// Else if own TU data index is free
ELSIF ZoneData.TransportControlData.TU_DataIndex = 0 THEN
	// Move TU data index from previous to own zone
	mTU_DataIndex := F_MoveTU_DataIndex(
							eFunctionNumber := PrevTransportData.eFunctionNumber,
							mZoneNumber     := PrevTransportData.ZoneNumber);

	// Update zone data
	ZoneData.TransportControlData.TU_DataIndex := mTU_DataIndex;
	ZoneData.TransportControlData.DataPresent := mTU_DataIndex <> 0;
	ZoneData.TransportControlData.NumberOfPresentTUs := 1;

	// Check if the TU data index is valid - if not, create a debug message
	IF mTU_DataIndex < 0 OR mTU_DataIndex > Conveyor.NUMBER_OF_TU_DATA THEN
		// debug message: '11-001-0095-01-1,  TU_DataIndex is out of range,  TU_DataIndex = 5000,  range = 0..1979'
		DebugMsg:= '';
		DebugMsg:= CONCAT(DebugMsg, Param.rSettings.ZoneName);
		DebugMsg:= CONCAT(DebugMsg, ',  TU_DataIndex is out of range');
		DebugMsg:= CONCAT(DebugMsg, DebugTextBlocks.TU_DATA_INDEX);
		DebugMsg:= CONCAT(DebugMsg, DINT_TO_STRING(mTU_DataIndex));
		DebugMsg:= CONCAT(DebugMsg, DebugTextBlocks.RANGE);
		DebugMsg:= CONCAT(DebugMsg, DINT_TO_STRING(Conveyor.NUMBER_OF_TU_DATA));
		fbDebugMsg.M_SendErrorMsg(DebugMsg);				  
		
	// Else if a valid TU data index is available check whether the index matches the expected position.
	// If not the TU index is incorrectly linked to multiple positions at the same time.
	ELSIF mTU_DataIndex <> 0 THEN
		mCurrentFunctionNumber := TU_Table.TU_DataTable[mTU_DataIndex].CurrentFunctionNumber;
		mCurrentZoneNumber := TU_Table.TU_DataTable[mTU_DataIndex].CurrentZoneNumber;
		
		// If function and zone number is valid
		IF mCurrentFunctionNumber <> 0 AND mCurrentZoneNumber <> 0 THEN
			// If current TU position is not previous zone
			IF mCurrentFunctionNumber <> PrevTransportData.eFunctionNumber OR mCurrentZoneNumber <> PrevTransportData.ZoneNumber THEN
				// debug message: '11-001-0095-01-1,  incorrectly linked TU_DataIndex to current TU position,  expected = 11-222-3333-44-5,  current = 99-9999-1979-01-9'
				DebugMsg:= '';
				DebugMsg:= CONCAT(DebugMsg, Param.rSettings.ZoneName);
				DebugMsg:= CONCAT(DebugMsg, ',  incorrectly linked TU_DataIndex to current TU position');
				DebugMsg:= CONCAT(DebugMsg, DebugTextBlocks.EXPECTED);
				DebugMsg:= CONCAT(DebugMsg, F_GetFunctionName(
												eFunctionNumber := PrevTransportData.eFunctionNumber,
												ZoneNumber := PrevTransportData.ZoneNumber));
				DebugMsg:= CONCAT(DebugMsg, DebugTextBlocks.CURRENT);
				DebugMsg:= CONCAT(DebugMsg, F_GetFunctionName(
												eFunctionNumber := mCurrentFunctionNumber,
												ZoneNumber := mCurrentZoneNumber));
				DebugMsg:= CONCAT(DebugMsg, F_CreateTU_DataString(mTU_DataIndex));
				fbDebugMsg.M_SendErrorMsg(DebugMsg);				  
			END_IF
		END_IF

		// Update currrent TU position
		TU_Table.TU_DataTable[mTU_DataIndex].CurrentFunctionNumber := Param.reFunctionNumber;
		TU_Table.TU_DataTable[mTU_DataIndex].CurrentZoneNumber := Param.ZoneNumber;
	END_IF

ELSE
	// Own TU data index is already used
	mTU_DataIndex := ZoneData.TransportControlData.TU_DataIndex;

	// Set error TU data index is not free
	F_SetError(
		ErrorType := E_ErrorType.ERROR,
		ErrorParam:= CONCAT('TU-DataIndex = ', DINT_TO_STRING(mTU_DataIndex)),
		ErrorMsg  := E_ErrorConv.TU_DATA_INDEX_NOT_FREE,
		ErrorData := ErrorData);
	
	// debug message: '11-001-0095-01-1,  own TU data index not free,  TU_DataIndex = 12345,  TuID = 112233,  AssignmentID = 12345678'
	DebugMsg:= '';
	DebugMsg:= CONCAT(DebugMsg, Param.rSettings.ZoneName);
	DebugMsg:= CONCAT(DebugMsg, ',  own TU data index not free');
	DebugMsg:= CONCAT(DebugMsg, F_CreateTU_DataString(mTU_DataIndex));
	fbDebugMsg.M_SendErrorMsg(DebugMsg);				  
	
	// Update number of present TUs
	ZoneData.TransportControlData.NumberOfPresentTUs := 1;
END_IF
{warning restore C0371}
END_METHOD

// Requests the routing service to retrieve next partner
METHOD PROTECTED M_RequestNext
(**************************************************************************************
 *  Application     :   BoxControl Framework
 *  Revision date   :   $Date: 2021-04-10 12:07:10 +0200 (lör, 10 apr 2021) $
 *  Author          :   CDC
 * ------------------------------------------------------------------------------------
 *  © Swisslog AG
 *  Swisslog is not liable for any usage of this source code that is not agreed 
 *  on between Swisslog and the other party. The mandatory legal liability remains 
 *  unaffected.
 * ------------------------------------------------------------------------------------
 *  Revision History: 
 *
 *  VERSION DATE         INITIALS     DESCRIPTION
 *  0.0     DD.MM.YYYY   (name)       (explain customized modifications)
 *
 **************************************************************************************)
VAR_INPUT
END_VAR
{warning disable C0371}
// If no next zone or function is available
IF NextTransportData.eFunctionNumber = E_FunctionNumber.F_BEGIN_FUNCTION AND
   Param.reNextFunctionNumber = E_FunctionNumber.F_BEGIN_FUNCTION THEN	
	fbRoutingServiceRetry(IN := FALSE);
	TransportTrspDataReq.RequestNextTransportData := TRUE;

// If the routing update is enable	
ELSIF Param.rSettings.EnableRoutingUpdate THEN
	// If the next function ist not fix
	IF Param.reSetFuncNextFuncNumber = E_FunctionNumber.F_BEGIN_FUNCTION
	   AND NOT NextTransportData.rTransportControlData.TransportActive THEN
		// If the transport does not start in a reasonable time, initiate routing update
		IF ZoneData.TransportControlData.eHandOverState = E_HandOverState.IDLE OR
		   ZoneData.TransportControlData.eHandOverState = E_HandOverState.READY THEN
			fbRoutingServiceRetry(IN := TRUE, PT := RECALL_SERVICE_TIMEOUT);
			IF fbRoutingServiceRetry.Q THEN
				fbRoutingServiceRetry(IN := FALSE);
				TransportTrspDataReq.DeleteNextTransportData := TRUE;
				TransportTrspDataReq.RequestNextTransportData := TRUE;
			END_IF
		ELSE
			fbRoutingServiceRetry(IN := FALSE);
		END_IF
	ELSE
		fbRoutingServiceRetry(IN := FALSE);
	END_IF
END_IF
{warning restore C0371}
END_METHOD

// Requests the merging service to retrieve prev partner
METHOD PROTECTED M_RequestPrev
(**************************************************************************************
 *  Application     :   BoxControl Framework
 *  Revision date   :   $Date: 2021-04-10 12:07:10 +0200 (lör, 10 apr 2021) $
 *  Author          :   CDC
 * ------------------------------------------------------------------------------------
 *  © Swisslog AG
 *  Swisslog is not liable for any usage of this source code that is not agreed 
 *  on between Swisslog and the other party. The mandatory legal liability remains 
 *  unaffected.
 * ------------------------------------------------------------------------------------
 *  Revision History: 
 *
 *  VERSION DATE         INITIALS     DESCRIPTION
 *  0.0     DD.MM.YYYY   (name)       (explain customized modifications)
 *
 **************************************************************************************)
VAR_INPUT
END_VAR
{warning disable C0371}
// If no previous zone or function is available
IF PrevTransportData.eFunctionNumber = E_FunctionNumber.F_BEGIN_FUNCTION AND
   Param.rePrevFunctionNumber = E_FunctionNumber.F_BEGIN_FUNCTION THEN	
	fbMergingServiceRetry(IN := FALSE);
	TransportTrspDataReq.RequestPrevTransportData := TRUE;


// If the previous function ist not fix
ELSIF Param.reSetFuncPrevFuncNumber = E_FunctionNumber.F_BEGIN_FUNCTION
   AND NOT PrevTransportData.rTransportControlData.TransportActive THEN
	// If the transport does not start in a reasonable time, initiate merging update
	IF ZoneData.TransportControlData.eTakeOverState = E_TakeOverState.IDLE OR
	   ZoneData.TransportControlData.eTakeOverState = E_TakeOverState.READY THEN
		fbMergingServiceRetry(IN := TRUE, PT := RECALL_SERVICE_TIMEOUT);
		IF fbMergingServiceRetry.Q THEN
			fbMergingServiceRetry(IN := FALSE);
			TransportTrspDataReq.DeletePrevTransportData := TRUE;
			TransportTrspDataReq.RequestPrevTransportData := TRUE;
		END_IF
	END_IF
END_IF
{warning restore C0371}
END_METHOD

METHOD M_SelectSensor : BOOL
(**************************************************************************************
 *  Application     :   BoxControl Framework
 *  Revision date   :   $Date: 2021-04-10 12:07:10 +0200 (lör, 10 apr 2021) $
 *  Author          :   CDC
 * ------------------------------------------------------------------------------------
 *  © Swisslog AG
 *  Swisslog is not liable for any usage of this source code that is not agreed 
 *  on between Swisslog and the other party. The mandatory legal liability remains 
 *  unaffected.
 * ------------------------------------------------------------------------------------
 *  Revision History: 
 *
 *  VERSION DATE         INITIALS     DESCRIPTION
 *  0.0     DD.MM.YYYY   (name)       (explain customized modifications)
 *
 **************************************************************************************)
VAR_INPUT
END_VAR
{warning disable C0371}
IF ZoneData.AddOn.Orders.UseOwnSensor OR NOT Param.rSettings.EnableAddOnSensor THEN
    ZoneOccupiedSignal := ZoneOccupied;
ELSE
    ZoneOccupiedSignal := ZoneData.AddOn.Orders.AddOnSensor;
END_IF
{warning restore C0371}
END_METHOD

// Starts the tracking of the leading edge arriving from prev zone
METHOD PROTECTED M_StartPositionTracking
(**************************************************************************************
 *  Application     :   BoxControl Framework
 *  Revision date   :   $Date: 2021-04-10 12:07:10 +0200 (lör, 10 apr 2021) $
 *  Author          :   CDC
 * ------------------------------------------------------------------------------------
 *  © Swisslog AG
 *  Swisslog is not liable for any usage of this source code that is not agreed 
 *  on between Swisslog and the other party. The mandatory legal liability remains 
 *  unaffected.
 * ------------------------------------------------------------------------------------
 *  Revision History: 
 *
 *  VERSION DATE         INITIALS     DESCRIPTION
 *  0.0     DD.MM.YYYY   (name)       (explain customized modifications)
 *
 **************************************************************************************)
VAR
	PresetDistance     			: DINT; // Present distance for tracking leading edge
END_VAR

// Set preset distance based on available previous position data	
IF PrevTransportData.rTransportControlData.TU_LeadingEdgePos <> 0 THEN
	PresetDistance := -(UINT_TO_DINT(PrevTransportParam.ZoneLength) - PrevTransportData.rTransportControlData.TU_LeadingEdgePos);
ELSE
	PresetDistance := -(UINT_TO_DINT(PrevTransportParam.ZoneEndLength) - PrevTransportParam.StopDelayDistance);
END_IF

// Start tracking 
fbTrackingLeadingEdge(Run := FALSE);

fbTrackingLeadingEdge(Run	:= TRUE,
		EncoderValueInc 	:= EncoderValue,
		MaxEncoderValueInc	:= MaxEncoderValue,
		RateIncPerMM		:= 1,
		SetPoint			:= UINT_TO_DINT(16#FFFF),
		StartPoint			:= PresetDistance);
END_METHOD

// Calculates the distance, the TU must at least travel to be considered plausible
METHOD PROTECTED M_TakeoverPlausibleDistance : DINT
(**************************************************************************************
 *  Application     :   BoxControl Framework
 *  Revision date   :   $Date: 2021-04-10 12:07:10 +0200 (lör, 10 apr 2021) $
 *  Author          :   CDC
 * ------------------------------------------------------------------------------------
 *  © Swisslog AG
 *  Swisslog is not liable for any usage of this source code that is not agreed 
 *  on between Swisslog and the other party. The mandatory legal liability remains 
 *  unaffected.
 * ------------------------------------------------------------------------------------
 *  Revision History: 
 *
 *  VERSION DATE         INITIALS     DESCRIPTION
 *  0.0     DD.MM.YYYY   (name)       (explain customized modifications)
 *
 **************************************************************************************)
VAR
	Temp		: DINT		:= 0;
END_VAR

// valid value given from config -> use this
IF Param.rSettings.TakeoverPlausibilityDistance <> 0 THEN
	M_TakeoverPlausibleDistance := Param.rSettings.TakeoverPlausibilityDistance;
	RETURN;
END_IF

// no, calculate it:
// distance between TU's leading edge to the border of the prev zone 
Temp:= PrevTransportParam.ZoneEndLength - PrevTransportParam.StopDelayDistance;

// adding the distance from begin of own zone to the sensor
Temp:= Temp + UINT_TO_DINT(TransportParam.ZoneLength) - TransportParam.ZoneEndLength;

// return reduced value to give space for tolerance
M_TakeoverPlausibleDistance:= Temp - DIST_TO_OCCUPIED;
END_METHOD

END_FUNCTION_BLOCK

// ---- 20_Product/10_BCF/11_Conv/12_E_Functions/10_Helper/F_AckAddon.TcPOU
FUNCTION F_AckAddon : BOOL
(**************************************************************************************
 * 	Application		:	BoxControl Framework
 *	Revision		:	$Revision: 404529 $
 *	Revision date	:	$Date: 2018-04-23 08:21:38 +0200 (Mo., 23 Apr 2018) $
 *	Last changed by	:	$Author: b7bolm $
 *	URL				:	$URL: http://almscdc.swisslog.com/repo/SWPD/Development/BoxControlFramework/20_Release/trunk/01_Software/BCF/BCF/JumpStart/20_Product/10_App/12_E_Functions/10_Lib/10_Conv/10_Functions/F_AckAddon.TcPOU $
 *
 *	Purpose			:	Send acknowledge to an addon.
 *						Return Ack successful.
 *
 * ------------------------------------------------------------------------------------
 *	Copyright Swisslog [IP AG], Switzerland. All rights reserved.
 * 
 * ------------------------------------------------------------------------------------
 *	
 * 	Revision History: 
 *
 * 	VERSION			DATE			INITIALS			DESCRIPTION
 *	0.1				01.01.2001		swl					Example
 *
 **************************************************************************************)
VAR_INPUT
	eFunctionNumber			: E_FunctionNumber; // Element function Number
END_VAR



// Check if function number is valid
IF eFunctionNumber > E_FunctionNumber.F_BEGIN_FUNCTION AND
   eFunctionNumber < E_FunctionNumber.F_END_FUNCTION THEN

	F_AckAddon := __ISVALIDREF(FunctionRegistry[eFunctionNumber].rFunction);
	
	// Check reference is valid
	IF F_AckAddon THEN
   		// Send Ack command
   		FunctionRegistry[eFunctionNumber].rFunction.M_AddOnAck();
	END_IF
END_IF

END_FUNCTION

// ---- 20_Product/10_BCF/11_Conv/12_E_Functions/10_Helper/F_CheckDestination.TcPOU
FUNCTION F_CheckDestination : BOOL
(**************************************************************************************
 * 	Application		:	BoxControl Framework
 *	Revision		:	$Revision: 404529 $
 *	Revision date	:	$Date: 2018-04-23 08:21:38 +0200 (Mo., 23 Apr 2018) $
 *	Last changed by	:	$Author: b7bolm $
 *	URL				:	$URL: http://almscdc.swisslog.com/repo/SWPD/Development/BoxControlFramework/20_Release/trunk/01_Software/BCF/BCF/JumpStart/20_Product/10_App/12_E_Functions/10_Lib/10_Conv/10_Functions/F_CheckDestination.TcPOU $
 *
 *	Purpose			:	Check if TU on a position consists of the desired destination
 ç						Result True = Destination found
 *
 * ------------------------------------------------------------------------------------
 *	Copyright Swisslog [IP AG], Switzerland. All rights reserved.
 * 
 * ------------------------------------------------------------------------------------
 *	
 * 	Revision History: 
 *
 * 	VERSION			DATE			INITIALS			DESCRIPTION
 *	0.1				01.01.2001		swl					Example
 *
 **************************************************************************************)
VAR_INPUT
	eFunctionNumber		: E_FunctionNumber; // Function number
	ZoneNumber			: INT; // ZoneNumber
	DestFunctionNumber	: E_FunctionNumber; // Destination function number
	DestZoneNumber		: INT; // Destination zone number
END_VAR

VAR
	TU_DataIndex		: DINT;
	Idx					: INT;
END_VAR

// Init
F_CheckDestination := FALSE;

// Validate inputs
IF eFunctionNumber > E_FunctionNumber.F_BEGIN_FUNCTION AND
   eFunctionNumber < E_FunctionNumber.F_END_FUNCTION AND
   ZoneNumber > 0 AND
   ZoneNumber <= Conveyor.NUMBER_OF_ZONES_PER_FUNCTION THEN
   	// If zone is valid and consists of a TU-Data index
	IF __ISVALIDREF(FunctionRegistry[eFunctionNumber].Zone[ZoneNumber].refZoneData) THEN
		TU_DataIndex := FunctionRegistry[eFunctionNumber].Zone[ZoneNumber].refZoneData.TransportControlData.TU_DataIndex;
		
		IF TU_DataIndex > 0 THEN
			// Search for destination
			FOR Idx := 1 TO Conveyor.NUMBER_OF_DESTINATIONS DO
				IF TU_DataTable[TU_DataIndex].Destination[Idx].eFunctionNumber = DestFunctionNumber AND
				   TU_DataTable[TU_DataIndex].Destination[Idx].ZoneNumber = DestZoneNumber THEN
				   // Destination found
				   F_CheckDestination := TRUE;
				   EXIT;
				END_IF
			END_FOR
		END_IF
	END_IF
END_IF

END_FUNCTION

// ---- 20_Product/10_BCF/11_Conv/12_E_Functions/10_Helper/F_GetAdjacentTransportData.TcPOU
FUNCTION F_GetAdjacentTransportData : ST_TransportData
(**************************************************************************************
 * 	Application		:	BoxControl Framework
 *	Revision		:	$Revision: 404529 $
 *	Revision date	:	$Date: 2018-04-23 08:21:38 +0200 (Mo., 23 Apr 2018) $
 *	Last changed by	:	$Author: b7bolm $
 *	URL				:	$URL: http://almscdc.swisslog.com/repo/SWPD/Development/BoxControlFramework/20_Release/trunk/01_Software/BCF/BCF/JumpStart/20_Product/10_App/12_E_Functions/10_Lib/10_Conv/10_Functions/F_GetAdjacentTransportData.TcPOU $
 *
 *	Purpose			:	Get adjacent zone
 *
 * ------------------------------------------------------------------------------------
 *	Copyright Swisslog [IP AG], Switzerland. All rights reserved.
 * 
 * ------------------------------------------------------------------------------------
 *	
 * 	Revision History: 
 *
 * 	VERSION			DATE			INITIALS			DESCRIPTION
 *	0.1				01.01.2001		swl					Example
 *
 **************************************************************************************)
VAR_INPUT
	eFunctionNumber			: E_FunctionNumber; // Element function Number
	eSourceFunctionNumber	: E_FunctionNumber; // Calling function number
END_VAR


// Check if function number is valid
IF eFunctionNumber > E_FunctionNumber.F_BEGIN_FUNCTION AND
   eFunctionNumber < E_FunctionNumber.F_END_FUNCTION THEN

	// Check reference is valid
	IF __ISVALIDREF(FunctionRegistry[eFunctionNumber].rFunction) THEN
   		// Return adjacent transport data
   		F_GetAdjacentTransportData := FunctionRegistry[eFunctionNumber].rFunction.M_GetTransportData(
											meFunctionNumber := eSourceFunctionNumber);
	END_IF
END_IF

END_FUNCTION

// ---- 20_Product/10_BCF/11_Conv/12_E_Functions/10_Helper/F_GetDestination.TcPOU
FUNCTION F_GetDestination : ST_PositionIdent
(**************************************************************************************
 * 	Application		:	BoxControl Framework
 *	Revision		:	$Revision: 404529 $
 *	Revision date	:	$Date: 2018-04-23 08:21:38 +0200 (Mo., 23 Apr 2018) $
 *	Last changed by	:	$Author: b7bolm $
 *	URL				:	$URL: http://almscdc.swisslog.com/repo/SWPD/Development/BoxControlFramework/20_Release/trunk/01_Software/BCF/BCF/JumpStart/20_Product/10_App/12_E_Functions/10_Lib/10_Conv/10_Functions/F_GetDestination.TcPOU $
 *
 *	Purpose			:	Gets the specified destination of a position
 *
 * ------------------------------------------------------------------------------------
 *	Copyright Swisslog [IP AG], Switzerland. All rights reserved.
 * 
 * ------------------------------------------------------------------------------------
 *	
 * 	Revision History: 
 *
 * 	VERSION			DATE			INITIALS			DESCRIPTION
 *	0.1				01.01.2001		swl					Example
 *
 **************************************************************************************)
VAR_INPUT
	eFunctionNumber		: E_FunctionNumber; // Function number
	ZoneNumber			: INT; // ZoneNumber
	DestinationIdx		: INT; // Which destination slot (Default 1)
END_VAR

VAR
	TU_DataIndex		: DINT;
END_VAR

// Init
F_GetDestination.eFunctionNumber := E_FunctionNumber.F_BEGIN_FUNCTION;
F_GetDestination.ZoneNumber	:= 0;

// Validate inputs
IF eFunctionNumber > E_FunctionNumber.F_BEGIN_FUNCTION AND
   eFunctionNumber < E_FunctionNumber.F_END_FUNCTION AND
   ZoneNumber > 0 AND
   ZoneNumber <= Conveyor.NUMBER_OF_ZONES_PER_FUNCTION THEN
   	// If zone is valid and consists of a TU-Data index
	IF __ISVALIDREF(FunctionRegistry[eFunctionNumber].Zone[ZoneNumber].refZoneData) THEN
		TU_DataIndex := FunctionRegistry[eFunctionNumber].Zone[ZoneNumber].refZoneData.TransportControlData.TU_DataIndex;
		// Return destination slot
		IF DestinationIdx > 0 AND DestinationIdx <= Conveyor.NUMBER_OF_DESTINATIONS THEN
			F_GetDestination.eFunctionNumber := TU_DataTable[TU_DataIndex].Destination[DestinationIdx].eFunctionNumber;
			F_GetDestination.ZoneNumber	:= TU_DataTable[TU_DataIndex].Destination[DestinationIdx].ZoneNumber;;
		END_IF
	END_IF
END_IF

END_FUNCTION

// ---- 20_Product/10_BCF/11_Conv/12_E_Functions/10_Helper/F_GetFunctionErrorData.TcPOU
FUNCTION F_GetFunctionErrorData : ST_FunctionErrorStruct
(**************************************************************************************
 * 	Application		:	BoxControl Framework
 *	Revision		:	$Revision: 404529 $
 *	Revision date	:	$Date: 2018-04-23 08:21:38 +0200 (Mo., 23 Apr 2018) $
 *	Last changed by	:	$Author: b7bolm $
 *	URL				:	$URL: http://almscdc.swisslog.com/repo/SWPD/Development/BoxControlFramework/20_Release/trunk/01_Software/BCF/BCF/JumpStart/20_Product/10_App/12_E_Functions/10_Lib/10_Conv/10_Functions/F_GetFunctionErrorData.TcPOU $
 *
 *	Purpose			:	Return function error data
 *
 * ------------------------------------------------------------------------------------
 *	Copyright Swisslog [IP AG], Switzerland. All rights reserved.
 * 
 * ------------------------------------------------------------------------------------
 *	
 * 	Revision History: 
 *
 * 	VERSION			DATE			INITIALS			DESCRIPTION
 *	0.1				01.01.2001		swl					Example
 *
 **************************************************************************************)
VAR_INPUT
	eFunctionNumber		: E_FunctionNumber; // Function number
END_VAR

// Check if function number is valid
IF eFunctionNumber > E_FunctionNumber.F_BEGIN_FUNCTION AND
   eFunctionNumber < E_FunctionNumber.F_END_FUNCTION THEN
  
	// Check reference is valid
	IF __ISVALIDREF(FunctionRegistry[eFunctionNumber].rFunctionData) THEN
   		// Return error data
   		F_GetFunctionErrorData := FunctionRegistry[eFunctionNumber].rFunctionData.ErrorData;
	END_IF
END_IF

END_FUNCTION

// ---- 20_Product/10_BCF/11_Conv/12_E_Functions/10_Helper/F_GetFunctionExternalErrorData.TcPOU
FUNCTION F_GetFunctionExternalErrorData : ST_ErrorDataSet
(**************************************************************************************
 * 	Application		:	BoxControl Framework
 *	Revision		:	$Revision: 404529 $
 *	Revision date	:	$Date: 2018-04-23 08:21:38 +0200 (Mo., 23 Apr 2018) $
 *	Last changed by	:	$Author: b7bolm $
 *	URL				:	$URL: http://almscdc.swisslog.com/repo/SWPD/Development/BoxControlFramework/20_Release/trunk/01_Software/BCF/BCF/JumpStart/20_Product/10_App/12_E_Functions/10_Lib/10_Conv/10_Functions/F_GetFunctionExternalErrorData.TcPOU $
 *
 *	Purpose			:	Return function external error data
 *
 * ------------------------------------------------------------------------------------
 *	Copyright Swisslog [IP AG], Switzerland. All rights reserved.
 * 
 * ------------------------------------------------------------------------------------
 *	
 * 	Revision History: 
 *
 * 	VERSION			DATE			INITIALS			DESCRIPTION
 *	0.1				01.01.2001		swl					Example
 *
 **************************************************************************************)
VAR_INPUT
	eFunctionNumber		: E_FunctionNumber; // Function number
END_VAR

// Check if function number is valid
IF eFunctionNumber > E_FunctionNumber.F_BEGIN_FUNCTION AND
   eFunctionNumber < E_FunctionNumber.F_END_FUNCTION THEN
  
	// Check reference is valid
	IF __ISVALIDREF(FunctionRegistry[eFunctionNumber].rFunctionData) THEN
   		// Return error data
   		F_GetFunctionExternalErrorData := FunctionRegistry[eFunctionNumber].rFunctionData.ErrorData.ExternalError;
	END_IF
END_IF

END_FUNCTION

// ---- 20_Product/10_BCF/11_Conv/12_E_Functions/10_Helper/F_GetFunctionInterface.TcPOU
FUNCTION F_GetFunctionInterface : ST_FunctionInterface
(**************************************************************************************
 * 	Application		:	BoxControl Framework
 *	Revision		:	$Revision: 404529 $
 *	Revision date	:	$Date: 2018-04-23 08:21:38 +0200 (Mo., 23 Apr 2018) $
 *	Last changed by	:	$Author: b7bolm $
 *	URL				:	$URL: http://almscdc.swisslog.com/repo/SWPD/Development/BoxControlFramework/20_Release/trunk/01_Software/BCF/BCF/JumpStart/20_Product/10_App/12_E_Functions/10_Lib/10_Conv/10_Functions/F_GetFunctionInterface.TcPOU $
 *
 *	Purpose			:	Returns function interface
 *
 * ------------------------------------------------------------------------------------
 *	Copyright Swisslog [IP AG], Switzerland. All rights reserved.
 * 
 * ------------------------------------------------------------------------------------
 *	
 * 	Revision History: 
 *
 * 	VERSION			DATE			INITIALS			DESCRIPTION
 *	0.1				01.01.2001		swl					Example
 *
 **************************************************************************************)
VAR_INPUT
	eFunctionNumber		: E_FunctionNumber; // Element function Number
END_VAR

// Check if function number is valid
IF eFunctionNumber > E_FunctionNumber.F_BEGIN_FUNCTION AND
   eFunctionNumber < E_FunctionNumber.F_END_FUNCTION THEN
  
   // Check reference is valid
   IF __ISVALIDREF(FunctionRegistry[eFunctionNumber].rFunction) THEN
	   
   		// Return function interface
   		F_GetFunctionInterface := FunctionRegistry[eFunctionNumber].rFunction.FunctionInterface;
   END_IF
END_IF

END_FUNCTION

// ---- 20_Product/10_BCF/11_Conv/12_E_Functions/10_Helper/F_GetFunctionInterlock.TcPOU
FUNCTION F_GetFunctionInterlock : ST_Interlock
(**************************************************************************************
 * 	Application		:	BoxControl Framework
 *	Revision		:	$Revision: 404529 $
 *	Revision date	:	$Date: 2018-04-23 08:21:38 +0200 (Mo., 23 Apr 2018) $
 *	Last changed by	:	$Author: b7bolm $
 *	URL				:	$URL: http://almscdc.swisslog.com/repo/SWPD/Development/BoxControlFramework/20_Release/trunk/01_Software/BCF/BCF/JumpStart/20_Product/10_App/12_E_Functions/10_Lib/10_Conv/10_Functions/F_GetFunctionInterlock.TcPOU $
 *
 *	Purpose			:	Returns function interlock structure
 *
 * ------------------------------------------------------------------------------------
 *	Copyright Swisslog [IP AG], Switzerland. All rights reserved.
 * 
 * ------------------------------------------------------------------------------------
 *	
 * 	Revision History: 
 *
 * 	VERSION			DATE			INITIALS			DESCRIPTION
 *	0.1				01.01.2001		swl					Example
 *
 **************************************************************************************)
VAR_INPUT
	eFunctionNumber			: E_FunctionNumber; // Element function Number
END_VAR

// Check if function number is valid
IF eFunctionNumber > E_FunctionNumber.F_BEGIN_FUNCTION AND
   eFunctionNumber < E_FunctionNumber.F_END_FUNCTION THEN
  
	// Check reference is valid
	IF __ISVALIDREF(FunctionRegistry[eFunctionNumber].rFunctionInterface) THEN
   		// Return function interlock
   		F_GetFunctionInterlock := FunctionRegistry[eFunctionNumber].rFunctionInterface.Out.Interlock;
	END_IF
END_IF

END_FUNCTION

// ---- 20_Product/10_BCF/11_Conv/12_E_Functions/10_Helper/F_GetFunctionOperationState.TcPOU
FUNCTION F_GetFunctionOperationState : ST_PositionState
(**************************************************************************************
 * 	Application		:	BoxControl Framework
 *	Revision		:	$Revision: 404529 $
 *	Revision date	:	$Date: 2018-04-23 08:21:38 +0200 (Mo., 23 Apr 2018) $
 *	Last changed by	:	$Author: b7bolm $
 *	URL				:	$URL: http://almscdc.swisslog.com/repo/SWPD/Development/BoxControlFramework/20_Release/trunk/01_Software/BCF/BCF/JumpStart/20_Product/10_App/12_E_Functions/10_Lib/10_Conv/10_Functions/F_GetFunctionOperationState.TcPOU $
 *
 *	Purpose			:	Returns function states
 *
 * ------------------------------------------------------------------------------------
 *	Copyright Swisslog [IP AG], Switzerland. All rights reserved.
 * 
 * ------------------------------------------------------------------------------------
 *	
 * 	Revision History: 
 *
 * 	VERSION			DATE			INITIALS			DESCRIPTION
 *	0.1				01.01.2001		swl					Example
 *
 **************************************************************************************)
VAR_INPUT
	eFunctionNumber			: E_FunctionNumber; // Element function Number
END_VAR

// Check if function number is valid
IF eFunctionNumber > E_FunctionNumber.F_BEGIN_FUNCTION AND
   eFunctionNumber < E_FunctionNumber.F_END_FUNCTION THEN
  
	// Check reference is valid
	IF __ISVALIDREF(FunctionRegistry[eFunctionNumber].rFunctionData) THEN
   		// Return function data
   		F_GetFunctionOperationState := FunctionRegistry[eFunctionNumber].rFunctionData.OperationState;
	END_IF
END_IF

END_FUNCTION

// ---- 20_Product/10_BCF/11_Conv/12_E_Functions/10_Helper/F_GetFunctionSettings.TcPOU
FUNCTION F_GetFunctionSettings : ST_CFG_Function
(**************************************************************************************
 * 	Application		:	BoxControl Framework
 *	Revision		:	$Revision: 404529 $
 *	Revision date	:	$Date: 2018-04-23 08:21:38 +0200 (Mo., 23 Apr 2018) $
 *	Last changed by	:	$Author: b7bolm $
 *	URL				:	$URL: http://almscdc.swisslog.com/repo/SWPD/Development/BoxControlFramework/20_Release/trunk/01_Software/BCF/BCF/JumpStart/20_Product/10_App/12_E_Functions/10_Lib/10_Conv/10_Functions/F_GetFunctionSettings.TcPOU $
 *
 *	Purpose			:	Function settings.
 *
 * ------------------------------------------------------------------------------------
 *	Copyright Swisslog [IP AG], Switzerland. All rights reserved.
 * 
 * ------------------------------------------------------------------------------------
 *	
 * 	Revision History: 
 *
 * 	VERSION			DATE			INITIALS			DESCRIPTION
 *	0.1				01.01.2001		swl					Example
 *
 **************************************************************************************)
VAR_INPUT
	eFunctionNumber		: E_FunctionNumber; // Function number
END_VAR

// If reference is valid
IF __ISVALIDREF(FunctionRegistry[eFunctionNumber].rSettingsFunction) THEN
	// Return base settings
	F_GetFunctionSettings := FunctionRegistry[eFunctionNumber].rSettingsFunction;
END_IF

END_FUNCTION

// ---- 20_Product/10_BCF/11_Conv/12_E_Functions/10_Helper/F_GetFunctionType.TcPOU
FUNCTION F_GetFunctionType : E_FunctionType;
(**************************************************************************************
 * 	Application		:	BoxControl Framework
 *	Revision		:	$Revision: 404529 $
 *	Revision date	:	$Date: 2018-04-23 08:21:38 +0200 (Mo., 23 Apr 2018) $
 *	Last changed by	:	$Author: b7bolm $
 *	URL				:	$URL: http://almscdc.swisslog.com/repo/SWPD/Development/BoxControlFramework/20_Release/trunk/01_Software/BCF/BCF/JumpStart/20_Product/10_App/12_E_Functions/10_Lib/10_Conv/10_Functions/F_GetFunctionType.TcPOU $
 *
 *	Purpose			:	Return function name
 *
 * ------------------------------------------------------------------------------------
 *	Copyright Swisslog [IP AG], Switzerland. All rights reserved.
 * 
 * ------------------------------------------------------------------------------------
 *	
 * 	Revision History: 
 *
 * 	VERSION			DATE			INITIALS			DESCRIPTION
 *	0.1				01.01.2001		swl					Example
 *
 **************************************************************************************)
VAR_INPUT
	eFunctionNumber		: E_FunctionNumber; // Function number
END_VAR

// Return function name
F_GetFunctionType := FunctionRegistry[eFunctionNumber].eFunctionType;

END_FUNCTION

// ---- 20_Product/10_BCF/11_Conv/12_E_Functions/10_Helper/F_GetZoneErrorData.TcPOU
FUNCTION F_GetZoneErrorData : ST_ZoneErrorStruct
(**************************************************************************************
 * 	Application		:	BoxControl Framework
 *	Revision		:	$Revision: 404529 $
 *	Revision date	:	$Date: 2018-04-23 08:21:38 +0200 (Mo., 23 Apr 2018) $
 *	Last changed by	:	$Author: b7bolm $
 *	URL				:	$URL: http://almscdc.swisslog.com/repo/SWPD/Development/BoxControlFramework/20_Release/trunk/01_Software/BCF/BCF/JumpStart/20_Product/10_App/12_E_Functions/10_Lib/10_Conv/10_Functions/F_GetZoneErrorData.TcPOU $
 *
 *	Purpose			:	Return zone error data
 *
 * ------------------------------------------------------------------------------------
 *	Copyright Swisslog [IP AG], Switzerland. All rights reserved.
 * 
 * ------------------------------------------------------------------------------------
 *	
 * 	Revision History: 
 *
 * 	VERSION			DATE			INITIALS			DESCRIPTION
 *	0.1				01.01.2001		swl					Example
 *
 **************************************************************************************)
VAR_INPUT
	eFunctionNumber		: E_FunctionNumber;
	ZoneNumber			: INT; 
END_VAR
VAR
	ZoneData			: ARRAY[1..NUMBER_OF_ZONES_PER_FUNCTION] OF ST_ZoneData; // all zone data
END_VAR


// Check if function number and zone is valid
IF eFunctionNumber > E_FunctionNumber.F_BEGIN_FUNCTION AND
   eFunctionNumber < E_FunctionNumber.F_END_FUNCTION AND
   ZoneNumber > 0 AND ZoneNumber <= NUMBER_OF_ZONES_PER_FUNCTION THEN
  
   IF __ISVALIDREF(FunctionRegistry[eFunctionNumber].Zone[ZoneNumber].refZoneData) THEN
		// Zone errordata
		F_GetZoneErrorData := FunctionRegistry[eFunctionNumber].Zone[ZoneNumber].refZoneData.ErrorData;
	END_IF
END_IF

END_FUNCTION

// ---- 20_Product/10_BCF/11_Conv/12_E_Functions/10_Helper/F_GetZoneExternErrorData.TcPOU
FUNCTION F_GetZoneExternErrorData : ST_ErrorDataSet
(**************************************************************************************
 * 	Application		:	BoxControl Framework
 *	Revision		:	$Revision: 404529 $
 *	Revision date	:	$Date: 2018-04-23 08:21:38 +0200 (Mo., 23 Apr 2018) $
 *	Last changed by	:	$Author: b7bolm $
 *	URL				:	$URL: http://almscdc.swisslog.com/repo/SWPD/Development/BoxControlFramework/20_Release/trunk/01_Software/BCF/BCF/JumpStart/20_Product/10_App/12_E_Functions/10_Lib/10_Conv/10_Functions/F_GetZoneExternErrorData.TcPOU $
 *
 *	Purpose			:	Return zone extern error data
 *
 * ------------------------------------------------------------------------------------
 *	Copyright Swisslog [IP AG], Switzerland. All rights reserved.
 * 
 * ------------------------------------------------------------------------------------
 *	
 * 	Revision History: 
 *
 * 	VERSION			DATE			INITIALS			DESCRIPTION
 *	0.1				01.01.2001		swl					Example
 *
 **************************************************************************************)
VAR_INPUT
	eFunctionNumber		: E_FunctionNumber;
	ZoneNumber			: INT; 
END_VAR
VAR
	ZoneData			: ARRAY[1..NUMBER_OF_ZONES_PER_FUNCTION] OF ST_ZoneData; // all zone data
END_VAR


// Check if function number and zone is valid
IF eFunctionNumber > E_FunctionNumber.F_BEGIN_FUNCTION AND
   eFunctionNumber < E_FunctionNumber.F_END_FUNCTION AND
   ZoneNumber > 0 AND ZoneNumber <= NUMBER_OF_ZONES_PER_FUNCTION THEN
  
   IF __ISVALIDREF(FunctionRegistry[eFunctionNumber].Zone[ZoneNumber].refZoneData) THEN
		// Zone errordata
		F_GetZoneExternErrorData := FunctionRegistry[eFunctionNumber].Zone[ZoneNumber].refZoneData.ErrorData.ExternalError;
	END_IF
END_IF

END_FUNCTION

// ---- 20_Product/10_BCF/11_Conv/12_E_Functions/10_Helper/F_GetZoneInterface.TcPOU
FUNCTION F_GetZoneInterface : ST_ZoneInterface
(**************************************************************************************
 * 	Application		:	BoxControl Framework
 *	Revision		:	$Revision: 404529 $
 *	Revision date	:	$Date: 2018-04-23 08:21:38 +0200 (Mo., 23 Apr 2018) $
 *	Last changed by	:	$Author: b7bolm $
 *	URL				:	$URL: http://almscdc.swisslog.com/repo/SWPD/Development/BoxControlFramework/20_Release/trunk/01_Software/BCF/BCF/JumpStart/20_Product/10_App/12_E_Functions/10_Lib/10_Conv/10_Functions/F_GetZoneInterface.TcPOU $
 *
 *	Purpose			:	Returns zones interface
 *
 * ------------------------------------------------------------------------------------
 *	Copyright Swisslog [IP AG], Switzerland. All rights reserved.
 * 
 * ------------------------------------------------------------------------------------
 *	
 * 	Revision History: 
 *
 * 	VERSION			DATE			INITIALS			DESCRIPTION
 *	0.1				01.01.2001		swl					Example
 *
 **************************************************************************************)
VAR_INPUT
	eFunctionNumber		: E_FunctionNumber; // Element function Number
	ZoneNumber			: INT; 
END_VAR

// Check if function number is valid
IF eFunctionNumber > E_FunctionNumber.F_BEGIN_FUNCTION AND
   eFunctionNumber < E_FunctionNumber.F_END_FUNCTION THEN

	// Check reference is valid
	IF __ISVALIDREF(FunctionRegistry[eFunctionNumber].rFunction) THEN
   		// Return zone interface
   		 F_GetZoneInterface := FunctionRegistry[eFunctionNumber].rFunction.ZoneInterface[ZoneNumber];
	END_IF
END_IF

END_FUNCTION

// ---- 20_Product/10_BCF/11_Conv/12_E_Functions/10_Helper/F_GetZonesCount.TcPOU
// function counts all used zones between this given limits
FUNCTION PUBLIC F_GetZonesCount : DWORD
(**************************************************************************************
 * Application   : BoxControl Framework
 * Revision date : $Date: 2013-09-23 11:26:06 +0200 (Wed, 23 Sep 2015) $
 * Author        : CDC
 * ------------------------------------------------------------------------------------
 * © Swisslog AG * Swisslog is not liable for any usage of this source code that is not agreed
 * on between Swisslog and the other party. The mandatory legal liability remains * unaffected.
 * ------------------------------------------------------------------------------------
 * Project revision history:
 *
 * VERSION DATE         INITIALS     DESCRIPTION
 * 0.0     DD.MM.YYYY   (name)       (explain customized modifications)
 *
 **************************************************************************************)

(************************************************************************************************************)
VAR_INPUT
	Start				: E_FunctionNumber				:= 0;	// limit for counting
	End					: E_FunctionNumber				:= 0;	// limit for counting
END_VAR

(************************************************************************************************************)
VAR
	FctNbr				: E_FunctionNumber				:= 0;
	StartFct			: E_FunctionNumber				:= 0;
	EndFct				: E_FunctionNumber				:= 0;
	Count				: DWORD							:= 0;
END_VAR


IF Start < E_FunctionNumber.F_BEGIN_FUNCTION THEN
	Start:= E_FunctionNumber.F_BEGIN_FUNCTION;
END_IF
IF Start > E_FunctionNumber.F_END_FUNCTION THEN
	Start:= E_FunctionNumber.F_END_FUNCTION;
END_IF
IF End < E_FunctionNumber.F_BEGIN_FUNCTION THEN
	End:= E_FunctionNumber.F_BEGIN_FUNCTION;
END_IF
IF End > E_FunctionNumber.F_END_FUNCTION THEN
	End:= E_FunctionNumber.F_END_FUNCTION;
END_IF

IF Start < End
THEN
	StartFct:= Start;
	EndFct:= End;
ELSIF  Start > End
THEN
	StartFct:= End;
	EndFct:= Start;
ELSE
	StartFct:= End;
	EndFct:= Start;
END_IF

Count:= 0;
FOR FctNbr:= StartFct TO EndFct DO
	IF FunctionRegistry[FctNbr].Enable THEN
		IF __ISVALIDREF(FunctionRegistry[FctNbr].rSettingsFunction) THEN
			Count:= Count + INT_TO_DWORD(FunctionRegistry[FctNbr].rSettingsFunction.NumberOfZones);
		END_IF
	END_IF
END_FOR

F_GetZonesCount:= Count;

END_FUNCTION

// ---- 20_Product/10_BCF/11_Conv/12_E_Functions/10_Helper/F_GetZonesData.TcPOU
FUNCTION F_GetZonesData : ARRAY[1..NUMBER_OF_ZONES_PER_FUNCTION] OF ST_ZoneData
(**************************************************************************************
 * 	Application		:	BoxControl Framework
 *	Revision		:	$Revision: 404529 $
 *	Revision date	:	$Date: 2018-04-23 08:21:38 +0200 (Mo., 23 Apr 2018) $
 *	Last changed by	:	$Author: b7bolm $
 *	URL				:	$URL: http://almscdc.swisslog.com/repo/SWPD/Development/BoxControlFramework/20_Release/trunk/01_Software/BCF/BCF/JumpStart/20_Product/10_App/12_E_Functions/10_Lib/10_Conv/10_Functions/F_GetZonesData.TcPOU $
 *
 *	Purpose			:	Returns external zones data
 *
 * ------------------------------------------------------------------------------------
 *	Copyright Swisslog [IP AG], Switzerland. All rights reserved.
 * 
 * ------------------------------------------------------------------------------------
 *	
 * 	Revision History: 
 *
 * 	VERSION			DATE			INITIALS			DESCRIPTION
 *	0.1				01.01.2001		swl					Example
 *
 **************************************************************************************)
VAR_INPUT
	eFunctionNumber			: E_FunctionNumber; // Element function Number
END_VAR


// Check if function number is valid
IF eFunctionNumber > E_FunctionNumber.F_BEGIN_FUNCTION AND
   eFunctionNumber < E_FunctionNumber.F_END_FUNCTION THEN
  
	// Check reference is valid
	IF __ISVALIDREF(FunctionRegistry[eFunctionNumber].rFunction) THEN
   		// Return zone data
   		F_GetZonesData := FunctionRegistry[eFunctionNumber].rFunction.ZoneData;
	END_IF
END_IF

END_FUNCTION

// ---- 20_Product/10_BCF/11_Conv/12_E_Functions/10_Helper/F_GetZonesInterface.TcPOU
FUNCTION F_GetZonesInterface : ARRAY[1..NUMBER_OF_ZONES_PER_FUNCTION] OF ST_ZoneInterface
(**************************************************************************************
 * 	Application		:	BoxControl Framework
 *	Revision		:	$Revision: 404529 $
 *	Revision date	:	$Date: 2018-04-23 08:21:38 +0200 (Mo., 23 Apr 2018) $
 *	Last changed by	:	$Author: b7bolm $
 *	URL				:	$URL: http://almscdc.swisslog.com/repo/SWPD/Development/BoxControlFramework/20_Release/trunk/01_Software/BCF/BCF/JumpStart/20_Product/10_App/12_E_Functions/10_Lib/10_Conv/10_Functions/F_GetZonesInterface.TcPOU $
 *
 *	Purpose			:	Returns zones interface
 *
 * ------------------------------------------------------------------------------------
 *	Copyright Swisslog [IP AG], Switzerland. All rights reserved.
 * 
 * ------------------------------------------------------------------------------------
 *	
 * 	Revision History: 
 *
 * 	VERSION			DATE			INITIALS			DESCRIPTION
 *	0.1				01.01.2001		swl					Example
 *
 **************************************************************************************)
VAR_INPUT
	eFunctionNumber			: E_FunctionNumber; // Element function Number
END_VAR


// Check if function number is valid
IF eFunctionNumber > E_FunctionNumber.F_BEGIN_FUNCTION AND
   eFunctionNumber < E_FunctionNumber.F_END_FUNCTION THEN

	// Check reference is valid
	IF __ISVALIDREF(FunctionRegistry[eFunctionNumber].rFunction) THEN
   		// Return zone interface
   		 F_GetZonesInterface := FunctionRegistry[eFunctionNumber].rFunction.ZoneInterface;
	END_IF
END_IF

END_FUNCTION

// ---- 20_Product/10_BCF/11_Conv/12_E_Functions/10_Helper/F_IsFunctionErrorPending.TcPOU
FUNCTION F_IsFunctionErrorPending : BOOL
(**************************************************************************************
 * 	Application		:	BoxControl Framework
 *	Revision		:	$Revision: 404529 $
 *	Revision date	:	$Date: 2018-04-23 08:21:38 +0200 (Mo., 23 Apr 2018) $
 *	Last changed by	:	$Author: b7bolm $
 *	URL				:	$URL: http://almscdc.swisslog.com/repo/SWPD/Development/BoxControlFramework/20_Release/trunk/01_Software/BCF/BCF/JumpStart/20_Product/10_App/12_E_Functions/10_Lib/10_Conv/10_Functions/F_IsFunctionErrorPending.TcPOU $
 *
 *	Purpose			:	Check if an error is pending on function and its containing zones
 *
 * ------------------------------------------------------------------------------------
 *	Copyright Swisslog [IP AG], Switzerland. All rights reserved.
 * 
 * ------------------------------------------------------------------------------------
 *	
 * 	Revision History: 
 *
 * 	VERSION			DATE			INITIALS			DESCRIPTION
 *	0.1				01.01.2001		swl					Example
 *
 **************************************************************************************)
VAR_INPUT
	eFunctionNumber		: E_FunctionNumber; // Function number
END_VAR

// Initialize
F_IsFunctionErrorPending := FALSE;

// Check if element number is valid
IF eFunctionNumber > E_FunctionNumber.F_BEGIN_FUNCTION AND
   eFunctionNumber < E_FunctionNumber.F_END_FUNCTION THEN

	// Check reference is valid
	IF __ISVALIDREF(FunctionRegistry[eFunctionNumber].rFunctionData) THEN
   		// Return error state
   		F_IsFunctionErrorPending := FunctionRegistry[eFunctionNumber].rFunctionData.ErrorData.Error.ErrorType = E_ErrorType.ERROR OR
									FunctionRegistry[eFunctionNumber].rFunctionData.ErrorData.ZoneErrorPending;
	END_IF
END_IF

END_FUNCTION

// ---- 20_Product/10_BCF/11_Conv/12_E_Functions/10_Helper/F_ResetExternalFunctionError.TcPOU
FUNCTION F_ResetExternalFunctionError : BOOL
(**************************************************************************************
 * 	Application		:	BoxControl Framework
 *	Revision		:	$Revision: 404529 $
 *	Revision date	:	$Date: 2018-04-23 08:21:38 +0200 (Mo., 23 Apr 2018) $
 *	Last changed by	:	$Author: b7bolm $
 *	URL				:	$URL: http://almscdc.swisslog.com/repo/SWPD/Development/BoxControlFramework/20_Release/trunk/01_Software/BCF/BCF/JumpStart/20_Product/10_App/12_E_Functions/10_Lib/10_Conv/10_Functions/F_ResetExternalFunctionError.TcPOU $
 *
 *	Purpose			:	Reset external error
 *						Add an External error, which will be reported over the configured
 *						position.
 *						
 *
 * ------------------------------------------------------------------------------------
 *	Copyright Swisslog [IP AG], Switzerland. All rights reserved.
 * 
 * ------------------------------------------------------------------------------------
 *	
 * 	Revision History: 
 *
 * 	VERSION			DATE			INITIALS			DESCRIPTION
 *	0.1				01.01.2001		swl					Example
 *
 **************************************************************************************)
VAR_INPUT
	eFunctionNumber : E_FunctionNumber; 
	ZoneNumber		: INT;
	Reset			: BOOL;
END_VAR


// Validate inputs
IF eFunctionNumber > E_FunctionNumber.F_BEGIN_FUNCTION THEN
	IF __ISVALIDREF(FunctionRegistry[eFunctionNumber].rFunction) THEN
		// Reset external error on instance
		FunctionRegistry[eFunctionNumber].rFunction.M_ResetExternalError(
			mZoneNumber := ZoneNumber,
			mReset := Reset);
	END_IF
END_IF

END_FUNCTION

// ---- 20_Product/10_BCF/11_Conv/12_E_Functions/10_Helper/F_ResetFunctionError.TcPOU
FUNCTION F_ResetFunctionError : BOOL
(**************************************************************************************
 * 	Application		:	BoxControl Framework
 *	Revision		:	$Revision: 404529 $
 *	Revision date	:	$Date: 2018-04-23 08:21:38 +0200 (Mo., 23 Apr 2018) $
 *	Last changed by	:	$Author: b7bolm $
 *	URL				:	$URL: http://almscdc.swisslog.com/repo/SWPD/Development/BoxControlFramework/20_Release/trunk/01_Software/BCF/BCF/JumpStart/20_Product/10_App/12_E_Functions/10_Lib/10_Conv/10_Functions/F_ResetFunctionError.TcPOU $
 *
 *	Purpose			:	Reset function errors
 *
 * ------------------------------------------------------------------------------------
 *	Copyright Swisslog [IP AG], Switzerland. All rights reserved.
 * 
 * ------------------------------------------------------------------------------------
 *	
 * 	Revision History: 
 *
 * 	VERSION			DATE			INITIALS			DESCRIPTION
 *	0.1				01.01.2001		swl					Example
 *
 **************************************************************************************)
VAR_INPUT
	eFunctionNumber		: E_FunctionNumber; // Function number
	ZoneNumber			: INT; // Zone number
	ResetAll			: BOOL; // Reset function and all zones
END_VAR

// Check if function number is valid
IF eFunctionNumber > E_FunctionNumber.F_BEGIN_FUNCTION AND
   eFunctionNumber < E_FunctionNumber.F_END_FUNCTION THEN
  
	// If reference is valid
	IF __ISVALIDREF(FunctionRegistry[eFunctionNumber].rFunction) THEN
		// Reset function
		FunctionRegistry[eFunctionNumber].rFunction.M_ResetError(
						mZoneNumber := ZoneNumber,
						mResetAll	:= ResetAll);
	END_IF
END_IF

END_FUNCTION

// ---- 20_Product/10_BCF/11_Conv/12_E_Functions/10_Helper/F_SetEnableHandOver.TcPOU
FUNCTION F_SetEnableHandOver : BOOL
(**************************************************************************************
 * 	Application		:	BoxControl Framework
 *	Revision		:	$Revision: 404529 $
 *	Revision date	:	$Date: 2018-04-23 08:21:38 +0200 (Mo., 23 Apr 2018) $
 *	Last changed by	:	$Author: b7bolm $
 *	URL				:	$URL: http://almscdc.swisslog.com/repo/SWPD/Development/BoxControlFramework/20_Release/trunk/01_Software/BCF/BCF/JumpStart/20_Product/10_App/12_E_Functions/10_Lib/10_Conv/10_Functions/F_SetEnableHandOver.TcPOU $
 *
 *	Purpose			:	Set enable handover
 *
 * ------------------------------------------------------------------------------------
 *	Copyright Swisslog [IP AG], Switzerland. All rights reserved.
 * 
 * ------------------------------------------------------------------------------------
 *	
 * 	Revision History: 
 *
 * 	VERSION			DATE			INITIALS			DESCRIPTION
 *	0.1				01.01.2001		swl					Example
 *
 **************************************************************************************)
VAR_INPUT
	eFunctionNumber	: E_FunctionNumber; // Function number of corresponding function
	ZoneNumber 	: INT; // Zone number
	Value		: BOOL;
END_VAR

// Check if function number is valid
IF eFunctionNumber > E_FunctionNumber.F_BEGIN_FUNCTION AND
   eFunctionNumber < E_FunctionNumber.F_END_FUNCTION THEN
  
	// Check reference is valid
	IF __ISVALIDREF(FunctionRegistry[eFunctionNumber].rFunction) THEN
   		// Return tu data index
   		F_SetEnableHandOver := FunctionRegistry[eFunctionNumber].rFunction.M_SetEnableHandOver(mZoneNumber:= ZoneNumber, mValue := Value);
	END_IF
END_IF

END_FUNCTION

// ---- 20_Product/10_BCF/11_Conv/12_E_Functions/10_Helper/F_SetEnableTakeOver.TcPOU
FUNCTION F_SetEnableTakeOver : BOOL
(**************************************************************************************
 * 	Application		:	BoxControl Framework
 *	Revision		:	$Revision: 404529 $
 *	Revision date	:	$Date: 2018-04-23 08:21:38 +0200 (Mo., 23 Apr 2018) $
 *	Last changed by	:	$Author: b7bolm $
 *	URL				:	$URL: http://almscdc.swisslog.com/repo/SWPD/Development/BoxControlFramework/20_Release/trunk/01_Software/BCF/BCF/JumpStart/20_Product/10_App/12_E_Functions/10_Lib/10_Conv/10_Functions/F_SetEnableTakeOver.TcPOU $
 *
 *	Purpose			:	Set enable takeover
 *
 * ------------------------------------------------------------------------------------
 *	Copyright Swisslog [IP AG], Switzerland. All rights reserved.
 * 
 * ------------------------------------------------------------------------------------
 *	
 * 	Revision History: 
 *
 * 	VERSION			DATE			INITIALS			DESCRIPTION
 *	0.1				01.01.2001		swl					Example
 *
 **************************************************************************************)
VAR_INPUT
	eFunctionNumber	: E_FunctionNumber; // Function number of corresponding function
	ZoneNumber 	: INT; // Zone number
	Value		: BOOL;
END_VAR

// Check if function number is valid
IF eFunctionNumber > E_FunctionNumber.F_BEGIN_FUNCTION AND
   eFunctionNumber < E_FunctionNumber.F_END_FUNCTION THEN

	// Check reference is valid
	IF __ISVALIDREF(FunctionRegistry[eFunctionNumber].rFunction) THEN
   		// Return tu data index
   		F_SetEnableTakeOver := FunctionRegistry[eFunctionNumber].rFunction.M_SetEnableTakeOver(mZoneNumber:= ZoneNumber, mValue := Value);
	END_IF
END_IF

END_FUNCTION

// ---- 20_Product/10_BCF/11_Conv/12_E_Functions/10_Helper/F_SetEnableTransport.TcPOU
FUNCTION F_SetEnableTransport : BOOL
(**************************************************************************************
 * 	Application		:	BoxControl Framework
 *	Revision		:	$Revision: 404529 $
 *	Revision date	:	$Date: 2018-04-23 08:21:38 +0200 (Mo., 23 Apr 2018) $
 *	Last changed by	:	$Author: b7bolm $
 *	URL				:	$URL: http://almscdc.swisslog.com/repo/SWPD/Development/BoxControlFramework/20_Release/trunk/01_Software/BCF/BCF/JumpStart/20_Product/10_App/12_E_Functions/10_Lib/10_Conv/10_Functions/F_SetEnableTransport.TcPOU $
 *
 *	Purpose			:	Set enable transport
 *
 * ------------------------------------------------------------------------------------
 *	Copyright Swisslog [IP AG], Switzerland. All rights reserved.
 * 
 * ------------------------------------------------------------------------------------
 *	
 * 	Revision History: 
 *
 * 	VERSION			DATE			INITIALS			DESCRIPTION
 *	0.1				01.01.2001		swl					Example
 *
 **************************************************************************************)
VAR_INPUT
	eFunctionNumber	: E_FunctionNumber; // Function number of corresponding function
	ZoneNumber 	: INT; // Zone number
	Value		: BOOL;
END_VAR

// Check if function number is valid
IF eFunctionNumber > E_FunctionNumber.F_BEGIN_FUNCTION AND
   eFunctionNumber < E_FunctionNumber.F_END_FUNCTION THEN
  
	// Check reference is valid
	IF __ISVALIDREF(FunctionRegistry[eFunctionNumber].rFunction) THEN
   		// Return tu data index
   		F_SetEnableTransport := FunctionRegistry[eFunctionNumber].rFunction.M_SetEnableTransport(mZoneNumber:= ZoneNumber, mValue := Value);
	END_IF
END_IF

END_FUNCTION

// ---- 20_Product/10_BCF/11_Conv/12_E_Functions/10_Helper/F_SetExternalFunctionError.TcPOU
FUNCTION F_SetExternalFunctionError : BOOL
(**************************************************************************************
 * 	Application		:	BoxControl Framework
 *	Revision		:	$Revision: 404529 $
 *	Revision date	:	$Date: 2018-04-23 08:21:38 +0200 (Mo., 23 Apr 2018) $
 *	Last changed by	:	$Author: b7bolm $
 *	URL				:	$URL: http://almscdc.swisslog.com/repo/SWPD/Development/BoxControlFramework/20_Release/trunk/01_Software/BCF/BCF/JumpStart/20_Product/10_App/12_E_Functions/10_Lib/10_Conv/10_Functions/F_SetExternalFunctionError.TcPOU $
 *
 *	Purpose			:	Set external error
 *						Add an External error, which will be reported over the configured
 *						position.
 *						
 *
 * ------------------------------------------------------------------------------------
 *	Copyright Swisslog [IP AG], Switzerland. All rights reserved.
 * 
 * ------------------------------------------------------------------------------------
 *	
 * 	Revision History: 
 *
 * 	VERSION			DATE			INITIALS			DESCRIPTION
 *	0.1				01.01.2001		swl					Example
 *
 **************************************************************************************)
VAR_INPUT
	eFunctionNumber : E_FunctionNumber; 
	ZoneNumber		: INT;
	ErrorType		: E_ErrorType; // Error message type
	ErrorParam		: STRING(System.ERROR_PARAM_STRINGLENGTH); // Error parameter
	ErrorMsg		: INT; // Error message as String (Will be mapped to error code)
END_VAR


// Validate inputs
IF eFunctionNumber > E_FunctionNumber.F_BEGIN_FUNCTION THEN
	IF __ISVALIDREF(FunctionRegistry[eFunctionNumber].rFunction) THEN
		// Set external error on instance
		FunctionRegistry[eFunctionNumber].rFunction.M_SetExternalError(
			mZoneNumber := ZoneNumber,
			mErrorType 	:= ErrorType,
			mErrorParam := ErrorParam,
			mErrorCode 	:= ErrorMsg);
	END_IF
END_IF

END_FUNCTION

// ---- 20_Product/10_BCF/11_Conv/12_E_Functions/10_Helper/F_StoppingDistance.TcPOU
FUNCTION F_StoppingDistance : UINT
(**************************************************************************************
 * 	Application		:	BoxControl Framework
 *	Revision		:	$Revision: 404529 $
 *	Revision date	:	$Date: 2018-04-23 08:21:38 +0200 (Mo., 23 Apr 2018) $
 *	Last changed by	:	$Author: b7bolm $
 *	URL				:	$URL: http://almscdc.swisslog.com/repo/SWPD/Development/BoxControlFramework/20_Release/trunk/01_Software/BCF/BCF/JumpStart/20_Product/10_App/12_E_Functions/10_Lib/10_Conv/10_Functions/F_StoppingDistance.TcPOU $
 *
 *	Purpose			:	Calculate stopping distance based on QB1 (distance until the TU is stopped in mm).
 *						
 *
 * ------------------------------------------------------------------------------------
 *	Copyright Swisslog [IP AG], Switzerland. All rights reserved.
 * 
 * ------------------------------------------------------------------------------------
 *	
 * 	Revision History: 
 *
 * 	VERSION			DATE			INITIALS			DESCRIPTION
 *	0.1				01.01.2001		swl					Example
 *
 **************************************************************************************)
VAR_INPUT
	CurrentSpeed : INT; // Current speed [mmm/s]
END_VAR
VAR
END_VAR

// Calculate distance besed on QB1 formula
F_StoppingDistance := LREAL_TO_UINT((((EXPT(CurrentSpeed,2) * MAX_LOADING * 50 / 2000) / (1.8 * 2))) / 1000);

END_FUNCTION

// ---- 20_Product/10_BCF/11_Conv/12_E_Functions/FB_FunctionConv.TcPOU
FUNCTION_BLOCK FB_FunctionConv EXTENDS FB_BaseObject
(**************************************************************************************
 * 	Application		:	BoxControl Framework
 *	Revision		:	$Revision: 475069 $
 *	Revision date	:	$Date: 2021-04-09 16:13:33 +0200 (fre, 09 apr 2021) $
 *	Last changed by	:	$Author: d7mangc $
 *	URL				:	$URL: http://almscdc.swisslog.com/repo/SWPD/Development/BoxControlFramework/20_Release/tags/R1.12.0/01_Software/BCF/BCF/JumpStart/20_Product/10_BCF/11_Conv/12_E_Functions/FB_FunctionConv.TcPOU $
 *
 *	Purpose			:	Base function.
 *
 * ------------------------------------------------------------------------------------
 *	Copyright Swisslog [IP AG], Switzerland. All rights reserved.
 * 
 * ------------------------------------------------------------------------------------
 *	
 * 	Revision History: 
 *
 * 	VERSION			DATE			INITIALS			DESCRIPTION
 *	0.1				01.01.2001		swl					Example
  *
 **************************************************************************************)
VAR_INPUT
	ConfigFunction			: ST_CFG_Function; // Base element function configuration 
	InhibitStopping			: BOOL; // Inhibit state change from Stopping to stop in order to finish an ongoing action
END_VAR

VAR
	FunctionBase			: ST_FunctionBase; // Summary of values used by framework internally
END_VAR

VAR PERSISTENT
	ITC						: ST_ITC_Function; // ITC
	FunctionData			: ST_FunctionData; // Function data - external read only 
	ZoneData				: ARRAY [1..NUMBER_OF_ZONES_PER_FUNCTION] OF ST_ZoneData; // Zone data
	FunctionInterface		: ST_FunctionInterface; // Element function interface - external read/write 
	ZoneInterface    		: ARRAY [1..NUMBER_OF_ZONES_PER_FUNCTION] OF ST_ZoneInterface; // Zone interface
	SettingsFunction		: ST_CFG_Function; // Base element function settings 
END_VAR

(**************************************************************************************************************
   Function - Body never called!
***************************************************************************************************************)
;

ACTION A_ErrorHandler:
(**************************************************************************************
 * 	NAME		A_ErrorHandling
 * 	FUNCTION	Handles element 
 **************************************************************************************)
 

(**************************************************************************************************************
  Monitor function errors
***************************************************************************************************************)
M_MonitorFunctionErrors();


(**************************************************************************************************************
  Monitor zone errors
***************************************************************************************************************)
M_MonitorZoneErrors();
END_ACTION

ACTION A_StateControl:
(**************************************************************************************
 * 	NAME		A_StateControl
 * 	FUNCTION	Handles internal states and mode
 **************************************************************************************)
 
(**************************************************************************************
   System state
***************************************************************************************)
FunctionData.OperationState.Info := FunctionInterface.In.Element.OperationState.Info;

FunctionData.OperationState.InitRelease := FunctionInterface.In.Element.OperationState.InitRelease;

 (**************************************************************************************
   Function mode
***************************************************************************************)
FunctionData.OperationState.eMode := FunctionInterface.In.Element.OperationState.eMode;

(**************************************************************************************
   Function states
***************************************************************************************)
CASE FunctionData.OperationState.eState OF
	
	(**************************************************************************************
   		UNKNOWN state
	***************************************************************************************)
	E_PositionState.UNKNOWN:
		// Update internal state
		FunctionData.OperationState.eLastState := FunctionData.OperationState.eState;
		FunctionData.OperationState.eState := E_PositionState.STOPPED;	

		
   	(**************************************************************************************
   		STOPPED state
	***************************************************************************************)
	E_PositionState.STOPPED:
		// When element is not stopping
		IF FunctionInterface.In.Element.OperationState.eState = E_PositionState.STARTED AND
		   FunctionInterface.In.Element.OperationState.eMode = E_PositionMode.AUTO_MODE AND
           FunctionData.Init THEN
			// Update internal state
			FunctionData.OperationState.eLastState := FunctionData.OperationState.eState;
			FunctionData.OperationState.eState := E_PositionState.STARTING;	
		END_IF
		
	(**************************************************************************************
   		STOPPING state
	***************************************************************************************)
	E_PositionState.STOPPING:
		// Wait until transport is stopped
		FunctionBase.AllZonesStopped  := TRUE;
		FunctionBase.LinkedFunctionStopped := TRUE;
        FOR FunctionBase.Idx := 1 TO SettingsFunction.NumberOfZones DO
			IF NOT ZoneData[FunctionBase.Idx].TransportControlData.Stopped THEN
				FunctionBase.AllZonesStopped  := FALSE;
			END_IF
		END_FOR
		
		// Check if linked function is already stopped
		IF SettingsFunction.FunctionLink.eFunctionNumber > E_FunctionNumber.F_BEGIN_FUNCTION THEN
			FunctionBase.OperatingState := F_GetFunctionOperationState(eFunctionNumber := SettingsFunction.FunctionLink.eFunctionNumber);

			IF FunctionBase.OperatingState.eState <> E_PositionState.STOPPED THEN
				FunctionBase.LinkedFunctionStopped := FALSE;
			END_IF
		END_IF
		
		// Check that function and own element is stopped
		IF FunctionInterface.In.Element.OperationState.eState = E_PositionState.STOPPED OR 
		   FunctionInterface.In.Element.OperationState.eMode <> E_PositionMode.AUTO_MODE OR 
		   (FunctionBase.AllZonesStopped AND FunctionBase.LinkedFunctionStopped AND NOT InhibitStopping) THEN
			// Goto Stopped
			FunctionData.OperationState.eLastState := FunctionData.OperationState.eState;
			FunctionData.OperationState.eState := E_PositionState.STOPPED;
		END_IF

	(**************************************************************************************
   		STARTING state
	***************************************************************************************)
	E_PositionState.STARTING:
		IF FunctionInterface.In.Element.OperationState.eState <> E_PositionState.STARTED OR 
           FunctionInterface.In.Element.OperationState.eMode <> E_PositionMode.AUTO_MODE THEN
		   	// Update internal state
			FunctionData.OperationState.eLastState := FunctionData.OperationState.eState;
			FunctionData.OperationState.eState := E_PositionState.STOPPED;	
		ELSE
			// Update internal state
			FunctionData.OperationState.eLastState := FunctionData.OperationState.eState;
			FunctionData.OperationState.eState := E_PositionState.STARTED;	
		END_IF
		
	(**************************************************************************************
   		STARTED state
	***************************************************************************************)
	E_PositionState.STARTED:
		IF FunctionInterface.In.Element.OperationState.eState = E_PositionState.STOPPING AND
           FunctionInterface.In.Element.OperationState.eMode = E_PositionMode.AUTO_MODE THEN
			// Update internal state
			FunctionData.OperationState.eLastState := FunctionData.OperationState.eState;
			FunctionData.OperationState.eState := E_PositionState.STOPPING;	
		ELSIF FunctionInterface.In.Element.OperationState.eState <> E_PositionState.STARTED OR 
              FunctionInterface.In.Element.OperationState.eMode <> E_PositionMode.AUTO_MODE THEN
			// Update internal state
			FunctionData.OperationState.eLastState := FunctionData.OperationState.eState;
			FunctionData.OperationState.eState := E_PositionState.STOPPED;	
		END_IF	
ELSE
	// Programming error
	DebugMsg := CONCAT(	'Programming error - Invalid state: ', INT_TO_STRING(FunctionData.OperationState.eState));
	fbDebugMsg.M_SendErrorMsg(DebugMsg);
END_CASE
END_ACTION

METHOD FB_init : BOOL

(********************************************************************************************************************************)
VAR_INPUT
	bInitRetains          : BOOL; // if TRUE, the retain variables are initialized (warm start / cold start)
	bInCopyCode           : BOOL;  // if TRUE, the instance afterwards gets moved into the copy code (online change)
END_VAR

// prepare empty values to be used for not-found or empty return values
FunctionBase.TransportDataEmpty.eFunctionNumber:= E_FunctionNumber.F_BEGIN_FUNCTION;
FunctionBase.TransportDataEmpty.ZoneNumber     := 0;
FunctionBase.TransportDataEmpty.rTransportControlData REF= FunctionBase.TransportControlDataEmpty;
FunctionBase.TransportDataEmpty.rSettings             REF= FunctionBase.ZoneSettingsEmpty;

FunctionBase.PrevTransportData:= FunctionBase.TransportDataEmpty;
FunctionBase.NextTransportData:= FunctionBase.TransportDataEmpty;
END_METHOD

METHOD M_AddOnAck : BOOL
(**************************************************************************************
 * 	Application		:	BoxControl Framework
 *	Revision		:	$Revision: 475069 $
 *	Revision date	:	$Date: 2021-04-09 16:13:33 +0200 (fre, 09 apr 2021) $
 *	Last changed by	:	$Author: d7mangc $
 *	URL				:	$URL: http://almscdc.swisslog.com/repo/SWPD/Development/BoxControlFramework/20_Release/tags/R1.12.0/01_Software/BCF/BCF/JumpStart/20_Product/10_BCF/11_Conv/12_E_Functions/FB_FunctionConv.TcPOU $
 *
 *	Purpose			:	Sends acknowledge command to addon
 *
 * ------------------------------------------------------------------------------------
 *	Copyright Swisslog [IP AG], Switzerland. All rights reserved.
 * 
 * ------------------------------------------------------------------------------------
 *	
 * 	Revision History: 
 *
 * 	VERSION			DATE			INITIALS			DESCRIPTION
 *	0.1				01.01.2001		swl					Example
 *
 **************************************************************************************)

// Set bit to inform the addon functionality was processed
FunctionBase.AddOnAck := TRUE;
END_METHOD

METHOD M_CloseAddOnLink : BOOL
(**************************************************************************************
 * 	Application		:	BoxControl Framework
 *	Revision		:	$Revision: 475069 $
 *	Revision date	:	$Date: 2021-04-09 16:13:33 +0200 (fre, 09 apr 2021) $
 *	Last changed by	:	$Author: d7mangc $
 *	URL				:	$URL: http://almscdc.swisslog.com/repo/SWPD/Development/BoxControlFramework/20_Release/tags/R1.12.0/01_Software/BCF/BCF/JumpStart/20_Product/10_BCF/11_Conv/12_E_Functions/FB_FunctionConv.TcPOU $
 *
 *	Purpose			:	Close link between Addon function and function
 *
 * ------------------------------------------------------------------------------------
 *	Copyright Swisslog [IP AG], Switzerland. All rights reserved.
 * 
 * ------------------------------------------------------------------------------------
 *	
 * 	Revision History: 
 *
 * 	VERSION			DATE			INITIALS			DESCRIPTION
 *	0.1				01.01.2001		swl					Example
 *
 **************************************************************************************)
VAR_INPUT
	eAddOnNumber		: E_FunctionNumber; // Function number
END_VAR
VAR
	mIdx				: INT; // Iterator
	mNextSlot			: INT; // Next slot
	mOldAddOnList		: ARRAY [1 .. NUMBER_OF_ADDON_FUNCTIONS] OF ST_AddonEntry; // Old function list
END_VAR
// Initialize
M_CloseAddOnLink := FALSE;
mNextSlot := 1;

// Check if element link is valid
IF eAddOnNumber > E_FunctionNumber.F_BEGIN_FUNCTION AND 
   eAddOnNumber < E_FunctionNumber.F_END_FUNCTION THEN
   
   // Clear incoming addon interface
   MEMSET(destAddr := ADR(FunctionInterface.In.AddOnOrder), fillByte := 0, n := SIZEOF(FunctionInterface.In.AddOnOrder));

   	// Go trough all slots
   	FOR mIdx := 1 TO NUMBER_OF_FUNCTIONS_PER_ELEMENT DO
		
		// Search registred function number
		IF FunctionData.MemberList.AddOnList[mIdx].eFunctionNumber = eAddOnNumber THEN
   			// Remove function 
			FunctionData.MemberList.AddOnList[mIdx].eFunctionNumber := E_FunctionNumber.F_BEGIN_FUNCTION;
			FunctionData.MemberList.AddOnList[mIdx].ZoneNumber := 0;

			// Element link closing was successfull
			M_CloseAddOnLink := TRUE;
		END_IF
   	END_FOR
	
	// Store old addon list
	mOldAddOnList := FunctionData.MemberList.AddOnList;
	
	// Remove gaps in addon list
   	FOR mIdx := 1 TO NUMBER_OF_ADDON_FUNCTIONS DO
		// If list index has a valid function number
		IF mOldAddOnList[mIdx].eFunctionNumber <> E_FunctionNumber.F_BEGIN_FUNCTION THEN
			// Store function in current list
			FunctionData.MemberList.AddOnList[mNextSlot].eFunctionNumber := mOldAddOnList[mIdx].eFunctionNumber;
			
			// Update index of current list
			mNextSlot := mNextSlot + 1;
		END_IF
   	END_FOR
	
	// Clear list
   	FOR mNextSlot := mNextSlot TO NUMBER_OF_FUNCTIONS_PER_ELEMENT DO
		// Clear entry
		FunctionData.MemberList.AddOnList[mNextSlot].eFunctionNumber := E_FunctionNumber.F_BEGIN_FUNCTION;
   	END_FOR
END_IF
END_METHOD

METHOD M_CreateAddOnLink : BOOL
(**************************************************************************************
 * 	Application		:	BoxControl Framework
 *	Revision		:	$Revision: 475069 $
 *	Revision date	:	$Date: 2021-04-09 16:13:33 +0200 (fre, 09 apr 2021) $
 *	Last changed by	:	$Author: d7mangc $
 *	URL				:	$URL: http://almscdc.swisslog.com/repo/SWPD/Development/BoxControlFramework/20_Release/tags/R1.12.0/01_Software/BCF/BCF/JumpStart/20_Product/10_BCF/11_Conv/12_E_Functions/FB_FunctionConv.TcPOU $
 *
 *	Purpose			:	Register an addon in function.
 *
 * ------------------------------------------------------------------------------------
 *	Copyright Swisslog [IP AG], Switzerland. All rights reserved.
 * 
 * ------------------------------------------------------------------------------------
 *	
 * 	Revision History: 
 *
 * 	VERSION			DATE			INITIALS			DESCRIPTION
 *	0.1				01.01.2001		swl					Example
 *
 **************************************************************************************)
VAR_INPUT
	eAddOnNumber		: E_FunctionNumber; // Function number
	ZoneNumber			: INT; // Zone number
END_VAR
VAR
	mIdx				: INT; // Iterator
END_VAR
// Initialize
M_CreateAddOnLink := FALSE;

// Check if addOn link is valid
IF eAddOnNumber > E_FunctionNumber.F_BEGIN_FUNCTION AND 
   eAddOnNumber < E_FunctionNumber.F_END_FUNCTION THEN
   
   	// Go trough all addOn slots
   	FOR mIdx := 1 TO NUMBER_OF_ADDON_FUNCTIONS DO
		
		// Search for free or an already registred slot for the desired addon function
		IF FunctionData.MemberList.AddOnList[mIdx].eFunctionNumber = E_FunctionNumber.F_BEGIN_FUNCTION OR 
		   FunctionData.MemberList.AddOnList[mIdx].eFunctionNumber = eAddOnNumber THEN
   			// Register addon
			FunctionData.MemberList.AddOnList[mIdx].eFunctionNumber := eAddOnNumber;
			FunctionData.MemberList.AddOnList[mIdx].ZoneNumber := ZoneNumber;
			
			// Registration was successfull
			M_CreateAddOnLink := TRUE;
			EXIT;
		END_IF
   	END_FOR
	
	// If error occured during registration
	IF NOT M_CreateAddOnLink THEN
		// No free slot found
		DebugMsg := 'No free addon registration slot found.';
		fbDebugMsg.M_SendErrorMsg(DebugMsg);
	END_IF
END_IF
END_METHOD

METHOD M_DeleteTU_DataIndex : BOOL
(**************************************************************************************
 * 	Application		:	BoxControl Framework
 *	Revision		:	$Revision: 475069 $
 *	Revision date	:	$Date: 2021-04-09 16:13:33 +0200 (fre, 09 apr 2021) $
 *	Last changed by	:	$Author: d7mangc $
 *	URL				:	$URL: http://almscdc.swisslog.com/repo/SWPD/Development/BoxControlFramework/20_Release/tags/R1.12.0/01_Software/BCF/BCF/JumpStart/20_Product/10_BCF/11_Conv/12_E_Functions/FB_FunctionConv.TcPOU $
 *
 *	Purpose			:	Delete TU Data index on position
 *
 * ------------------------------------------------------------------------------------
 *	Copyright Swisslog [IP AG], Switzerland. All rights reserved.
 * 
 * ------------------------------------------------------------------------------------
 *	
 * 	Revision History: 
 *
 * 	VERSION			DATE			INITIALS			DESCRIPTION
 *	0.1				01.01.2001		swl					Example
 *
 **************************************************************************************)
VAR_INPUT
	mZoneNumber		: INT; // Zone number
	mTU_DataIndex	: DINT; // Tu index to delete
	mInit			: BOOL; // Initialize position afterwards
END_VAR
// Initialize
M_DeleteTU_DataIndex := FALSE;

// Zone number valid
IF mZoneNumber > 0 AND mZoneNumber <= SettingsFunction.NumberOfZones THEN
	// TU Index is equal to the current
	IF mTU_DataIndex = ZoneData[mZoneNumber].TransportControlData.TU_DataIndex THEN
		// Clear
		ZoneData[mZoneNumber].TransportControlData.TU_DataIndex := 0;
		ZoneData[mZoneNumber].TransportControlData.DataPresent := FALSE;
		
		// Init requested
		IF mInit THEN
			ZoneData[mZoneNumber].Init := FALSE;
		END_IF
		
		// Delete successful
		M_DeleteTU_DataIndex := TRUE;
		
		// BCFD-11639 - POR0 - Position Cleared Report sent without TU-ID	
		// included in BCF 1.16
		// Save data from the last TU for the position clear report
		M_SaveDataTU_ZoneLeft (mZoneNumber, mTU_DataIndex); 
	END_IF
END_IF
END_METHOD

METHOD M_FindTU_DataIndex : BOOL
(**************************************************************************************
 * 	Application		:	BoxControl Framework
 *	Revision		:	$Revision: 475069 $
 *	Revision date	:	$Date: 2021-04-09 16:13:33 +0200 (fre, 09 apr 2021) $
 *	Last changed by	:	$Author: d7mangc $
 *	URL				:	$URL: http://almscdc.swisslog.com/repo/SWPD/Development/BoxControlFramework/20_Release/tags/R1.12.0/01_Software/BCF/BCF/JumpStart/20_Product/10_BCF/11_Conv/12_E_Functions/FB_FunctionConv.TcPOU $
 *
 *	Purpose			:	Checks if a position consists of specific TU_DataIndex.
 *						mZoneNumber 0 = search in whole position
 *						This method can be overwritten for example in a Belt, to give 
 *						access to internal TU index structures.
 *
 * ------------------------------------------------------------------------------------
 *	Copyright Swisslog [IP AG], Switzerland. All rights reserved.
 * 
 * ------------------------------------------------------------------------------------
 *	
 * 	Revision History: 
 *
 * 	VERSION			DATE			INITIALS			DESCRIPTION
 *	0.1				01.01.2001		swl					Example
 *
 **************************************************************************************)
VAR_INPUT
	mZoneNumber		: INT; // Check zone number, 0 = check all
	mTU_DataIndex	: DINT; // Searched TU index
END_VAR

VAR
	mIdx			: INT; // Iterator
END_VAR
// Initialize
M_FindTU_DataIndex := FALSE;

// If Zone index is in a specific range 
IF mZoneNumber > 0 AND mZoneNumber <= SettingsFunction.NumberOfZones THEN
	// Check for index
	M_FindTU_DataIndex := ZoneData[mZoneNumber].TransportControlData.TU_DataIndex = mTU_DataIndex;
ELSIF mZoneNumber = 0 THEN
	// Check all configured zones
	FOR mIdx := 1 TO SettingsFunction.NumberOfZones DO
		M_FindTU_DataIndex := ZoneData[mIdx].TransportControlData.TU_DataIndex = mTU_DataIndex;
		// If an index was found -> Exit
		IF M_FindTU_DataIndex THEN
			RETURN;
		END_IF
	END_FOR
END_IF
END_METHOD

// Copies AddOnOrders into the function interface
METHOD PROTECTED M_GetAddOnOrder
(**************************************************************************************
 *  Application     :   BoxControl Framework
 *  Revision date   :   $Date: 2021-04-09 16:13:33 +0200 (fre, 09 apr 2021) $
 *  Author          :   CDC
 * ------------------------------------------------------------------------------------
 *  © Swisslog AG
 *  Swisslog is not liable for any usage of this source code that is not agreed 
 *  on between Swisslog and the other party. The mandatory legal liability remains 
 *  unaffected.
 * ------------------------------------------------------------------------------------
 *  Revision History: 
 *
 *  VERSION DATE         INITIALS     DESCRIPTION
 *  0.0     DD.MM.YYYY   (name)       (explain customized modifications)
 *
 **************************************************************************************)
VAR
	mIdx					: INT;	// Iterator
	meAddOnFunctionNumber	: E_FunctionNumber;	// Function numebr
	mControlledZoneNumber	: INT;	// zone number
END_VAR

// Go through all addon members
FOR mIdx := 1 TO NUMBER_OF_ADDON_FUNCTIONS DO

	// If a valid addon is registerd
	IF FunctionData.MemberList.AddOnList[mIdx].eFunctionNumber > E_FunctionNumber.F_BEGIN_FUNCTION AND
	   FunctionData.MemberList.AddOnList[mIdx].eFunctionNumber < E_FunctionNumber.F_END_FUNCTION THEN

	   meAddOnFunctionNumber := FunctionData.MemberList.AddOnList[mIdx].eFunctionNumber;
	   
	   // Check if a valid reference is available for that function and the function is initialized
		IF __ISVALIDREF(FunctionRegistry[meAddOnFunctionNumber].rFunctionInterface) AND
		   F_IsFunctionInitialized(meAddOnFunctionNumber) THEN
			mControlledZoneNumber:= FunctionData.MemberList.AddOnList[mIdx].ZoneNumber;
			// Store them internally
			FunctionInterface.In.AddOnOrder[mIdx].eFunctionNumber := meAddOnFunctionNumber;
			FunctionInterface.In.AddOnOrder[mIdx].ZoneNumber      := mControlledZoneNumber;
			// data from controlling add on
			FunctionInterface.In.AddOnOrder[mIdx].eFunctionType   := FunctionRegistry[meAddOnFunctionNumber].eFunctionType;
			FunctionInterface.In.AddOnOrder[mIdx].Orders          := FunctionRegistry[meAddOnFunctionNumber].rFunction.M_GetOutAddOnOrders(eFunctionNumber:= SettingsFunction.eFunctionNumber,
																																			ZoneNumber    := mControlledZoneNumber);
		ELSE
			MEMSET(destAddr := ADR(FunctionInterface.In.AddOnOrder[mIdx]), fillByte := 0, n := SIZEOF(FunctionInterface.In.AddOnOrder[mIdx]));
		END_IF
	ELSE
		// No valid addon functions
		EXIT;
	END_IF
END_FOR
END_METHOD

METHOD PROTECTED M_GetElementStates 
(**************************************************************************************
 * 	Application		:	BoxControl Framework
 *	Revision		:	$Revision: 475069 $
 *	Revision date	:	$Date: 2021-04-09 16:13:33 +0200 (fre, 09 apr 2021) $
 *	Last changed by	:	$Author: d7mangc $
 *	URL				:	$URL: http://almscdc.swisslog.com/repo/SWPD/Development/BoxControlFramework/20_Release/tags/R1.12.0/01_Software/BCF/BCF/JumpStart/20_Product/10_BCF/11_Conv/12_E_Functions/FB_FunctionConv.TcPOU $
 *
 *	Purpose			:	Get states of corresponding element
 *
 * ------------------------------------------------------------------------------------
 *	Copyright Swisslog [IP AG], Switzerland. All rights reserved.
 * 
 * ------------------------------------------------------------------------------------
 *	
 * 	Revision History: 
 *
 * 	VERSION			DATE			INITIALS			DESCRIPTION
 *	0.1				01.01.2001		swl					Example
 *
 **************************************************************************************)
VAR
	mIdx					: INT; // Iterator
	meElementNumber			: E_ElementNumber; 
END_VAR

// If element link is valid
IF SettingsFunction.eElementLink > E_ElementNumber.E_BEGIN_ELEMENT AND
   SettingsFunction.eElementLink < E_ElementNumber.E_END_ELEMENT THEN
  
	meElementNumber := SettingsFunction.eElementLink;
	
   // Check element is initialized and has valid references
   IF __ISVALIDREF(ElementRegistry[meElementNumber].rElementData) AND
      __ISVALIDREF(ElementRegistry[meElementNumber].rElementInterface) AND
      F_IsElementInitialized(meElementNumber) THEN
   		// Return 
		FunctionInterface.In.Element.OperationState := ElementRegistry[meElementNumber].rElementData.OperationState;
		FunctionInterface.In.Element.State := ElementRegistry[meElementNumber].rElementInterface.Out.State;
   ELSE
	    MEMSET(destAddr := ADR(FunctionInterface.In.Element), fillByte := 0, n := SIZEOF(FunctionInterface.In.Element));
   END_IF
END_IF
END_METHOD

METHOD PROTECTED M_GetNextTransportData : REFERENCE TO ST_TransportData
(**************************************************************************************
 * 	Application		:	BoxControl Framework
 *	Revision		:	$Revision: 475069 $
 *	Revision date	:	$Date: 2021-04-09 16:13:33 +0200 (fre, 09 apr 2021) $
 *	Last changed by	:	$Author: d7mangc $
 *	URL				:	$URL: http://almscdc.swisslog.com/repo/SWPD/Development/BoxControlFramework/20_Release/tags/R1.12.0/01_Software/BCF/BCF/JumpStart/20_Product/10_BCF/11_Conv/12_E_Functions/FB_FunctionConv.TcPOU $
 *
 *	Purpose			:	Get transport data for next zone
 *
 * ------------------------------------------------------------------------------------
 *	Copyright Swisslog [IP AG], Switzerland. All rights reserved.
 * 
 * ------------------------------------------------------------------------------------
 *	
 * 	Revision History: 
 *
 * 	VERSION			DATE			INITIALS			DESCRIPTION
 *	0.1				01.01.2001		swl					Example
 *
 **************************************************************************************)
VAR_INPUT
	mZoneNumber : INT; // Number of the zone
END_VAR

VAR
	meFunctionNumber : E_FunctionNumber;
	NextZoneNumber : INT;
END_VAR
(*
* Check where the next zone is located at depending also on the flow direction (1 to x or x to 1) and number of the zones the function has.
* Then return reference to the TransportData in that zone. If next was not found, return reference to the empty TransportData.
*)
//If there was no decision, return empty reference
M_GetNextTransportData REF= FunctionBase.TransportDataEmpty;
		
IF (mZoneNumber = 1 AND SettingsFunction.FlowDirectionREV)
	OR (mZoneNumber = SettingsFunction.NumberOfZones AND NOT SettingsFunction.FlowDirectionREV) THEN	
	// If the function number is valid
	IF FunctionInterface.In.eNextFunctionNumber > E_FunctionNumber.F_BEGIN_FUNCTION AND
	   FunctionInterface.In.eNextFunctionNumber < E_FunctionNumber.F_END_FUNCTION THEN
	    
		meFunctionNumber := FunctionInterface.In.eNextFunctionNumber;

		// If the reference is valid and the function is initialized
		IF __ISVALIDREF(FunctionRegistry[meFunctionNumber].rFunction)  AND
		   F_IsFunctionInitialized(meFunctionNumber) THEN
			// Return adjacent transport data of the adjacent function
			M_GetNextTransportData REF= FunctionRegistry[meFunctionNumber].rFunction
											.M_GetTransportData(meFunctionNumber := SettingsFunction.eFunctionNumber);
		END_IF
		
	// If the function number points to an external interface
	ELSIF FunctionInterface.In.eNextFunctionNumber > E_FunctionNumber.F_BEGIN_EXTERN_FUNCTION AND
		  FunctionInterface.In.eNextFunctionNumber < E_FunctionNumber.F_END_EXTERN_FUNCTION THEN
		// Check interface is valid
		IF __QUERYINTERFACE(fbSTI_Channels[FunctionInterface.In.eNextFunctionNumber].Instance,FunctionBase.STI_Instance) THEN
			// Return adjacent transport data of the adjacent external function
			M_GetNextTransportData REF= fbSTI_Channels[FunctionInterface.In.eNextFunctionNumber].Instance.M_GetTransportData();
		END_IF
	END_IF
ELSE
	//Calculate the number of the next zone depending on the flow direction
	IF SettingsFunction.FlowDirectionREV THEN 
		NextZoneNumber := mZoneNumber - 1;
	ELSE
		NextZoneNumber := mZoneNumber + 1;
	END_IF

	FunctionBase.NextTransportData.eFunctionNumber := SettingsFunction.eFunctionNumber;
	FunctionBase.NextTransportData.ZoneNumber := NextZoneNumber;	
	FunctionBase.NextTransportData.rTransportControlData REF= ZoneData[NextZoneNumber].TransportControlData;
	FunctionBase.NextTransportData.rSettings REF= SettingsFunction.Zone[NextZoneNumber];	
	M_GetNextTransportData REF= FunctionBase.NextTransportData;
END_IF
END_METHOD

// Returns the orders to control a linked function/zone
METHOD PROTECTED M_GetOutAddOnOrders : ST_AddOnOrders
(**************************************************************************************
 *  Application     :   BoxControl Framework
 *  Revision date   :   $Date: 2021-04-09 16:13:33 +0200 (fre, 09 apr 2021) $
 *  Author          :   CDC
 * ------------------------------------------------------------------------------------
 *  © Swisslog AG
 *  Swisslog is not liable for any usage of this source code that is not agreed 
 *  on between Swisslog and the other party. The mandatory legal liability remains 
 *  unaffected.
 * ------------------------------------------------------------------------------------
 *  Revision History: 
 *
 *  VERSION DATE         INITIALS     DESCRIPTION
 *  0.0     DD.MM.YYYY   (name)       (explain customized modifications)
 *
 **************************************************************************************)
VAR_INPUT
	eFunctionNumber		: E_FunctionNumber	:= 0;	// Function number to be controlled
	ZoneNumber			: INT				:= 0;	// zone number to be controlled
END_VAR

M_GetOutAddOnOrders:= FunctionInterface.Out.AddOnOrders;
END_METHOD

METHOD PROTECTED M_GetPreviousTransportData: REFERENCE TO ST_TransportData
(**************************************************************************************
 * 	Application		:	BoxControl Framework
 *	Revision		:	$Revision: 475069 $
 *	Revision date	:	$Date: 2021-04-09 16:13:33 +0200 (fre, 09 apr 2021) $
 *	Last changed by	:	$Author: d7mangc $
 *	URL				:	$URL: http://almscdc.swisslog.com/repo/SWPD/Development/BoxControlFramework/20_Release/tags/R1.12.0/01_Software/BCF/BCF/JumpStart/20_Product/10_BCF/11_Conv/12_E_Functions/FB_FunctionConv.TcPOU $
 *
 *	Purpose			:	Get transport data from previous zone
 *
 * ------------------------------------------------------------------------------------
 *	Copyright Swisslog [IP AG], Switzerland. All rights reserved.
 * 
 * ------------------------------------------------------------------------------------
 *	
 * 	Revision History: 
 *
 * 	VERSION			DATE			INITIALS			DESCRIPTION
 *	0.1				01.01.2001		swl					Example
 *  0.2				27.02.2020		jmu					Refactored
 *
 **************************************************************************************)
VAR_INPUT
	mZoneNumber 	: INT; // Number of the zone
END_VAR

VAR
	meFunctionNumber	: E_FunctionNumber;
	PreviousZoneNumber : INT;
END_VAR
(*
* Check where the previous zone is located at depending also on the flow direction (1 to x or x to 1) and number of the zones the function has.
* Then return reference to the TransportData in that zone. If previous was not found, return reference to the empty TransportData.
*)
//If there was no decision, return empty reference
M_GetPreviousTransportData REF= FunctionBase.TransportDataEmpty;
		
IF (mZoneNumber = 1 AND NOT SettingsFunction.FlowDirectionREV)
	OR (mZoneNumber = SettingsFunction.NumberOfZones AND SettingsFunction.FlowDirectionREV) THEN	
	// If the function number is valid
	IF FunctionInterface.In.ePrevFunctionNumber > E_FunctionNumber.F_BEGIN_FUNCTION AND
	   FunctionInterface.In.ePrevFunctionNumber < E_FunctionNumber.F_END_FUNCTION THEN
	    
		meFunctionNumber := FunctionInterface.In.ePrevFunctionNumber;

		// If the reference is valid and the function is initialized
		IF __ISVALIDREF(FunctionRegistry[meFunctionNumber].rFunction)  AND
		   F_IsFunctionInitialized(meFunctionNumber) THEN
			// Return adjacent transport data of the adjacent function
			M_GetPreviousTransportData REF= FunctionRegistry[meFunctionNumber].rFunction
											.M_GetTransportData(meFunctionNumber := SettingsFunction.eFunctionNumber);
		END_IF
		
	// If the function number points to an external interface
	ELSIF FunctionInterface.In.ePrevFunctionNumber > E_FunctionNumber.F_BEGIN_EXTERN_FUNCTION AND
		  FunctionInterface.In.ePrevFunctionNumber < E_FunctionNumber.F_END_EXTERN_FUNCTION THEN
		// Check interface is valid
		IF __QUERYINTERFACE(fbSTI_Channels[FunctionInterface.In.ePrevFunctionNumber].Instance,FunctionBase.STI_Instance) THEN
			// Return adjacent transport data of the adjacent external function
			M_GetPreviousTransportData REF= fbSTI_Channels[FunctionInterface.In.ePrevFunctionNumber].Instance.M_GetTransportData();
		END_IF
	END_IF
ELSE
	//Calculate the number of the previous zone depending on the flow direction
	IF SettingsFunction.FlowDirectionREV THEN 
		PreviousZoneNumber := mZoneNumber + 1;
	ELSE
		PreviousZoneNumber := mZoneNumber - 1;
	END_IF

	FunctionBase.PrevTransportData.eFunctionNumber := SettingsFunction.eFunctionNumber;
	FunctionBase.PrevTransportData.ZoneNumber := PreviousZoneNumber;	
	FunctionBase.PrevTransportData.rTransportControlData REF= ZoneData[PreviousZoneNumber].TransportControlData;
	FunctionBase.PrevTransportData.rSettings REF= SettingsFunction.Zone[PreviousZoneNumber];	
	M_GetPreviousTransportData REF= FunctionBase.PrevTransportData;
END_IF
END_METHOD

METHOD PROTECTED M_GetTransportControlParam : REFERENCE TO ST_TransportControlParam
(**************************************************************************************
 * 	Application		:	BoxControl Framework
 *	Revision		:	$Revision: 475069 $
 *	Revision date	:	$Date: 2021-04-09 16:13:33 +0200 (fre, 09 apr 2021) $
 *	Last changed by	:	$Author: d7mangc $
 *	URL				:	$URL: http://almscdc.swisslog.com/repo/SWPD/Development/BoxControlFramework/20_Release/tags/R1.12.0/01_Software/BCF/BCF/JumpStart/20_Product/10_BCF/11_Conv/12_E_Functions/FB_FunctionConv.TcPOU $
 *
 *	Purpose			:	Get transport control parameter
 *
 * ------------------------------------------------------------------------------------
 *	Copyright Swisslog [IP AG], Switzerland. All rights reserved.
 * 
 * ------------------------------------------------------------------------------------
 *	
 * 	Revision History: 
 *
 * 	VERSION			DATE			INITIALS			DESCRIPTION
 *	0.1				01.01.2001		swl					Example
 *
 **************************************************************************************)
VAR_INPUT
	mZoneNumber : INT; // Number of the zone
END_VAR

// Return function number
FunctionBase.TransportControlParam.reFunctionNumber REF= SettingsFunction.eFunctionNumber;
// Return function state
FunctionBase.TransportControlParam.rOperationState REF= FunctionData.OperationState;

// Return previous function number
FunctionBase.TransportControlParam.rePrevFunctionNumber REF= FunctionInterface.In.ePrevFunctionNumber;
// Return next function number
FunctionBase.TransportControlParam.reNextFunctionNumber REF= FunctionInterface.In.eNextFunctionNumber;

// Return zone enable
FunctionBase.TransportControlParam.rZoneEnable REF= ZoneInterface[mZoneNumber].In.Enable;
// Return external zone enable
FunctionBase.TransportControlParam.rExternalZoneEnable REF= ZoneInterface[mZoneNumber].In.ZoneEnable;

// Return settings prev/next function number
FunctionBase.TransportControlParam.reSetFuncPrevFuncNumber REF= SettingsFunction.ePrevFunctionNumber;
FunctionBase.TransportControlParam.reSetFuncNextFuncNumber REF= SettingsFunction.eNextFunctionNumber;

// Return zone number
FunctionBase.TransportControlParam.ZoneNumber := mZoneNumber;
// Return zone settings
FunctionBase.TransportControlParam.rSettings REF= SettingsFunction.Zone[mZoneNumber];

M_GetTransportControlParam REF= FunctionBase.TransportControlParam;
END_METHOD

METHOD M_GetTransportData : REFERENCE TO ST_TransportData
(**************************************************************************************
 * 	Application		:	BoxControl Framework
 *	Revision		:	$Revision: 475069 $
 *	Revision date	:	$Date: 2021-04-09 16:13:33 +0200 (fre, 09 apr 2021) $
 *	Last changed by	:	$Author: d7mangc $
 *	URL				:	$URL: http://almscdc.swisslog.com/repo/SWPD/Development/BoxControlFramework/20_Release/tags/R1.12.0/01_Software/BCF/BCF/JumpStart/20_Product/10_BCF/11_Conv/12_E_Functions/FB_FunctionConv.TcPOU $
 *
 *	Purpose			:	Get adjacent zone
 *
 * ------------------------------------------------------------------------------------
 *	Copyright Swisslog [IP AG], Switzerland. All rights reserved.
 * 
 * ------------------------------------------------------------------------------------
 *	
 * 	Revision History: 
 *
 * 	VERSION			DATE			INITIALS			DESCRIPTION
 *	0.1				01.01.2001		swl					Example
 *
 **************************************************************************************)
VAR_INPUT
	meFunctionNumber : E_FunctionNumber; // Own element function number
END_VAR
(*
Initialize
Reference points initialy to an empty struct, to ensure
always a valid reference, even no decision could be made.
*)
M_GetTransportData REF= FunctionBase.TransportDataEmpty;

// If the function number is valid
IF meFunctionNumber > F_BEGIN_FUNCTION THEN
	// If the requesting function is the previous function
	IF meFunctionNumber = FunctionInterface.In.ePrevFunctionNumber THEN
		// If the flow direction is forward
		IF NOT SettingsFunction.FlowDirectionREV THEN
			// Return the transport data of the first zone
			FunctionBase.TransportData.eFunctionNumber := SettingsFunction.eFunctionNumber;
			FunctionBase.TransportData.ZoneNumber := 1;
			FunctionBase.TransportData.rSettings REF= SettingsFunction.Zone[1];
			FunctionBase.TransportData.rTransportControlData REF= ZoneData[1].TransportControlData;
			M_GetTransportData REF= FunctionBase.TransportData;
		ELSE
			// If the zone number is valid
			IF SettingsFunction.NumberOfZones > 0 THEN
				// Return the transport data of the last zone
				FunctionBase.TransportData.eFunctionNumber := SettingsFunction.eFunctionNumber;
				FunctionBase.TransportData.ZoneNumber := SettingsFunction.NumberOfZones;
				FunctionBase.TransportData.rSettings REF= SettingsFunction.Zone[SettingsFunction.NumberOfZones];
				FunctionBase.TransportData.rTransportControlData REF= ZoneData[SettingsFunction.NumberOfZones].TransportControlData;	
				M_GetTransportData REF= FunctionBase.TransportData;
			END_IF	
		END_IF
	
	// If the requesting function is the next function
	ELSIF meFunctionNumber = FunctionInterface.In.eNextFunctionNumber THEN
		
		// If the flow direction is forward
		IF NOT SettingsFunction.FlowDirectionREV THEN
			// If the zone number is valid
			IF SettingsFunction.NumberOfZones > 0 THEN
				// Return the transport data of the last zone
				FunctionBase.TransportData.eFunctionNumber := SettingsFunction.eFunctionNumber;
				FunctionBase.TransportData.ZoneNumber := SettingsFunction.NumberOfZones;
				FunctionBase.TransportData.rSettings REF= SettingsFunction.Zone[SettingsFunction.NumberOfZones];
				FunctionBase.TransportData.rTransportControlData REF= ZoneData[SettingsFunction.NumberOfZones].TransportControlData;
				M_GetTransportData REF= FunctionBase.TransportData;
			END_IF
		ELSE
			// Return the transport data of the first zone
			FunctionBase.TransportData.eFunctionNumber := SettingsFunction.eFunctionNumber;
			FunctionBase.TransportData.ZoneNumber := 1;
			FunctionBase.TransportData.rSettings REF= SettingsFunction.Zone[1];
			FunctionBase.TransportData.rTransportControlData REF= ZoneData[1].TransportControlData;
			M_GetTransportData REF= FunctionBase.TransportData;
		END_IF
	END_IF
END_IF
END_METHOD

METHOD M_InitFunction : BOOL
(**************************************************************************************
 * 	Application		:	BoxControl Framework
 *	Revision		:	$Revision: 475069 $
 *	Revision date	:	$Date: 2021-04-09 16:13:33 +0200 (fre, 09 apr 2021) $
 *	Last changed by	:	$Author: d7mangc $
 *	URL				:	$URL: http://almscdc.swisslog.com/repo/SWPD/Development/BoxControlFramework/20_Release/tags/R1.12.0/01_Software/BCF/BCF/JumpStart/20_Product/10_BCF/11_Conv/12_E_Functions/FB_FunctionConv.TcPOU $
 *
 *	Purpose			:	Initialize base functionality of function.
 *
 * ------------------------------------------------------------------------------------
 *	Copyright Swisslog [IP AG], Switzerland. All rights reserved.
 * 
 * ------------------------------------------------------------------------------------
 *	
 * 	Revision History: 
 *
 * 	VERSION			DATE			INITIALS			DESCRIPTION
 *	0.1				01.01.2001		swl					Example
 *
 **************************************************************************************)
VAR_INPUT
	mReset			: BOOL; // Reset initialization flag
END_VAR

VAR
	mName			: T_MaxString; // Alpha numeric string only
	mIdx			: INT; // Iterator
	eFunctionNumber	: E_FunctionNumber; 
	eElementNumber	: E_ElementNumber;
END_VAR

// If the init was requested
IF mReset THEN
	// Inform the bottom function to initialize
	FunctionData.Init := FALSE;
	// Reset values and load config
	M_PreInit();
ELSE
	(**************************************************************************************
   		Initialize & Register
	***************************************************************************************)
	// Load basic configuration to settings
	SettingsFunction := ConfigFunction;
	
	// Remove non alpha numeric signs
	mName := F_ReduceToAlphaNumeric(InputString := SettingsFunction.FunctionName);

	// Update Registry reference with HashCode
	FunctionRegistry[SettingsFunction.eFunctionNumber].HashCode := F_CreateHashCode(InputString := mName);
	
	// Update Registry reference with name
	FunctionRegistry[SettingsFunction.eFunctionNumber].FunctionName := SettingsFunction.FunctionName;
	
	// Update Registry function type
	FunctionRegistry[SettingsFunction.eFunctionNumber].eFunctionType := SettingsFunction.eFunctionType;
	
	// Register and initialize all zones
	FOR mIdx := 1 TO NUMBER_OF_ZONES_PER_FUNCTION DO
		// Build name without alpha numerics
		mName := F_ReduceToAlphaNumeric(InputString := SettingsFunction.Zone[mIdx].ZoneName);
		
		// Initialize
		ZoneData[mIdx].AddOn.NoAddons := TRUE;
		ZoneData[mIdx].AddOn.Orders.Enable := TRUE;
		ZoneData[mIdx].AddOn.Orders.DataReady := TRUE;
		ZoneData[mIdx].AddOn.Orders.EnableHandover := TRUE;
		ZoneData[mIdx].AddOn.Orders.EnableTakeover := TRUE;
		ZoneData[mIdx].AddOn.Orders.TU_DataIndex := 0;
		
		// Register
		FunctionRegistry[SettingsFunction.eFunctionNumber].Zone[mIdx].ZoneName := SettingsFunction.Zone[mIdx].ZoneName;
		FunctionRegistry[SettingsFunction.eFunctionNumber].Zone[mIdx].HashCode := F_CreateHashCode(InputString := mName);
	END_FOR
	
	(**************************************************************************************
   		AddOn Register
	***************************************************************************************)
	
	// If Addon function link is available
	IF SettingsFunction.FunctionLink.eFunctionNumber < E_FunctionNumber.F_END_FUNCTION AND
       SettingsFunction.FunctionLink.eFunctionNumber > E_FunctionNumber.F_BEGIN_FUNCTION THEN
	   
		// Create addon link
		eFunctionNumber := SettingsFunction.FunctionLink.eFunctionNumber;
		
		// Is this reference valid
		IF __ISVALIDREF(FunctionRegistry[eFunctionNumber].rFunction) THEN
			// Create AddOn link
			FunctionRegistry[eFunctionNumber].rFunction.M_CreateAddOnLink(
										eAddOnNumber := SettingsFunction.eFunctionNumber,
										ZoneNumber	 := SettingsFunction.FunctionLink.ZoneNumber);
		END_IF
	END_IF
	
	
	(**************************************************************************************
   		Element register (Mandatory)
	***************************************************************************************)
	
	// Check if element link is valid
	IF SettingsFunction.eElementLink > E_ElementNumber.E_BEGIN_ELEMENT AND 
	   SettingsFunction.eElementLink < E_ElementNumber.E_END_ELEMENT THEN
		
	   	// Close old addon link
		eElementNumber := SettingsFunction.eElementLink;
		
		// Is reference valid
		IF __ISVALIDREF(ElementRegistry[eElementNumber].rElement) THEN
			// Register function in element
			M_InitFunction := ElementRegistry[eElementNumber].rElement.M_CreateElementLink(SettingsFunction.eFunctionNumber);
		END_IF
	END_IF
	
